      AN #s_Receive_Data_Outf.Itm_Data.Process_1.Screening_Not_Required;
      A #s_Receive_Data_Outf.Itm_Data.HBS_Record.PEN_Process_1.Result_Pending;
      A(;
      L "DB_HBS_List".HBS[#s_Receive_Data_Outf.Itm_Data.LNK_Record.HBS].LNK;// nlpcanh //#s_Receive_Data_Outf.Itm_Data.HBS_Record.PEN_General.HBA_LNK
      L #s_Receive_Data_Outf.Itm_Data.LNK;
      ==I;
      );
      A(;
      L #s_Receive_Data_Outf.Itm_Data.HBS_Record.PEN_Process_1.Screen_Result.Pseudo_ID;
      L #s_ISD_ID_Tracking.Data_10.BHS_Pseudo_Bag_ID;
      ==D;
      );
      S #s_Receive_Data_Outf.Itm_Data.Process_1.Screening_Pending;
      S #s_Receive_Data_Outf.Screening_Pending;// If a certain process contains the pseudo which is sent by the EDS, while "result expected": item is pending

IB01:      A #s_Receive_Data_Outf.EDS_Tracking.Trk_Lost_Result_Pending;
      JCN IB99;
//// [CPH] If lost in tracking inside the machine, do not expect/accept any further decisions
////      SET
////      S     #s_Receive_Data_Outf.Itm_Data.Process_1.Screening_Pending
////      S     #s_Receive_Data_Outf.Screening_Pending

IB99:      NOP 0;
NETWORK
TITLE = JA: Update GENERAL local records (HBS/LIC) at outfeed
//Local records will be updated to reflect the current bag status.
      A #s_OS_Receive_Bag_Data;// Bag tracking was restored (outfeed)
      A #s_Receive_Data_Outf.Tracking_Restored;// Check HBS record
      JCN JA99;

      L #i_HBS_ID;
      T #t_Last_Location;

      CALL "FC_Write_Dint_Record"
      (  i_Record_Number             := #s_Receive_Data_Outf.Itm_Data.LNK_Record.ECS ,
         i_P_DINT_Record             := "DB_UDT_ECS_Record".CIR.Last_Location ,
         i_DB                        := "DB_ECS_List" ,
         i_DINT                      := #t_Last_Location ,
         i_DB_Event_Num              := #t_DB_Event_Num_Object
      );

      A #s_Receive_Data_Outf.Screening_Pending;
      JCN JA99;

      A #s_Receive_Data_Outf.HBS_Record_Present;
      JCN JA01;

      CALL "FC_Read_ANY_Record"
      (  i_Record_Number             := #s_Receive_Data_Outf.Itm_Data.LNK_Record.HBS ,
         i_ANY_Data_Record           := "DB_UDT_HBS_Record".PEN_General ,
         i_ANY_Data                  := #s_Receive_Data_Outf.Itm_Data.HBS_Record.PEN_General ,
         i_DB                        := "DB_HBS_List" ,
         i_DB_Event_Num              := #t_DB_Event_Num_Object
      );

      JU JA99;

JA01:      CALL "FC_Generator_LNK"
      (  i_LNK                       := #s_Receive_Data_Outf.Itm_Data.LNK ,
         i_DB_List                   := #t_DB_HBS_List_Num ,
         i_Default_Record            := #i_Default_Record_Outf ,
         i_DB_Event_Num              := #t_DB_Event_Num_Object ,
         o_LNK                       := #t_INT_not_used
      );

      CALL "FC_Read_Int_Record"
      (  i_Record_Number             := #s_Receive_Data_Outf.Itm_Data.LNK ,
         i_P_INT_Record              := "DB_UDT_LNK_Record".HBS ,
         i_DB                        := "DB_LNK_List" ,
         i_DB_Event_Num              := #t_DB_Event_Num_Object ,
         o_INT                       := #s_Receive_Data_Outf.Itm_Data.LNK_Record.HBS
      );

      CALL "FC_Read_ANY_Record"
      (  i_Record_Number             := #s_Receive_Data_Outf.Itm_Data.LNK_Record.HBS ,
         i_ANY_Data_Record           := "DB_UDT_HBS_Record" ,
         i_ANY_Data                  := #s_Receive_Data_Outf.Itm_Data.HBS_Record ,
         i_DB                        := "DB_HBS_List" ,
         i_DB_Event_Num              := #t_DB_Event_Num_Object
      );

      L #s_Receive_Data_Outf.Itm_Data.LNK_Record.HBS;
      L 0;
      >I;
      S #s_Receive_Data_Outf.HBS_Record_Present;
      JCN JA99;// Creation succeeded

      SET;
      R #s_Receive_Data_Outf.Itm_Data.HBS_Record.PEN_General.Item_Lost;
      S #s_Receive_Data_Outf.Init_HBS_Record;

      L 0;
      T #s_Receive_Data_Outf.Itm_Data.HBS_Record.PEN_General.AreaID_Receive;

      CALL "FC_Write_ANY_Record"// Attach to bag
      (  i_Record_Number             := #s_Receive_Data_Outf.Itm_Data.LNK_Record.HBS ,
         i_ANY_Data_Record           := "DB_UDT_HBS_Record".PEN_General ,
         i_ANY_Data                  := #s_Receive_Data_Outf.Itm_Data.HBS_Record.PEN_General ,
         i_DB                        := "DB_HBS_List" ,
         i_DB_Event_Num              := #t_DB_Event_Num_Object
      );

      A #s_Receive_Data_Outf.New_LNK_Created;
      JCN JA99;// If new LNK with HBS was created: store HBS number in lookup table

      L #s_EDS_Pseudo_Lookup.Write_Position_Lookup_T;
      JL JA10;
      JU JA11;
      JU JA12;
      JU JA13;
      JU JA14;
      JU JA15;
JA10:      JU JA99;
JA11:      L #s_Receive_Data_Outf.Itm_Data.LNK_Record.HBS;
      T #s_EDS_Pseudo_Lookup.HBS_Lookup_Table[0];
      JU JA20;
JA12:      L #s_Receive_Data_Outf.Itm_Data.LNK_Record.HBS;
      T #s_EDS_Pseudo_Lookup.HBS_Lookup_Table[1];
      JU JA20;
JA13:      L #s_Receive_Data_Outf.Itm_Data.LNK_Record.HBS;
      T #s_EDS_Pseudo_Lookup.HBS_Lookup_Table[2];
      JU JA20;
JA14:      L #s_Receive_Data_Outf.Itm_Data.LNK_Record.HBS;
      T #s_EDS_Pseudo_Lookup.HBS_Lookup_Table[3];
      JU JA20;
JA15:      L #s_Receive_Data_Outf.Itm_Data.LNK_Record.HBS;
      T #s_EDS_Pseudo_Lookup.HBS_Lookup_Table[4];

JA20:      L #s_EDS_Pseudo_Lookup.Write_Position_Lookup_T;
      L 1;
      +I;
      T #s_EDS_Pseudo_Lookup.Write_Position_Lookup_T;

      L #s_EDS_Pseudo_Lookup.Write_Position_Lookup_T;
      L 4;
      >I;
      JCN JA99;

      L 0;
      T #s_EDS_Pseudo_Lookup.Write_Position_Lookup_T;
JA99:      NOP 0;
NETWORK
TITLE = JB: Update PROCESS_1 local records (HBS/LIC) at outfeed
      A #s_OS_Receive_Bag_Data;
      JCN JB99;

      A #s_Receive_Data_Outf.New_LNK_Created;
      AN #s_Receive_Data_Outf.LIC_Missing;
      JCN JB01;// If LIC is available and a new records was generated: attach pseudo, else: continue HBS record update

      CALL "FC_Write_Dint_Record"// Write pseudo to LIC
      (  i_Record_Number             := #s_Receive_Data_Outf.Itm_Data.LNK_Record.LIC ,
         i_P_DINT_Record             := "DB_UDT_LIC_Record".BIR.Process_1.Pseudo_ID ,
         i_DB                        := "DB_LIC_List" ,
         i_DINT                      := #s_PseudoId_To_Use_At_Exit , //#s_ISD_ID_Tracking.Data_10.BHS_Pseudo_Bag_ID
         i_DB_Event_Num              := #t_DB_Event_Num_Object
      );

JB01:      A #s_Receive_Data_Outf.Screening_Pending;
      A #s_Receive_Data_Outf.HBS_Record_Present;
      JCN JB99;// If new data prepared: create records and check if HBS record update is required

      A #s_Receive_Data_Outf.Init_HBS_Record;
      JCN JB02;

      SET;
      R #s_Receive_Data_Outf.Itm_Data.HBS_Record.PEN_Process_1.Machine_Result_Rcvd;
      R #s_Receive_Data_Outf.Itm_Data.HBS_Record.PEN_Process_1.Operator_Result_Rcvd;
      R #s_Receive_Data_Outf.Itm_Data.HBS_Record.PEN_Process_1.Result_Pending;
      R #s_Receive_Data_Outf.Itm_Data.HBS_Record.PEN_Process_1.Update_Send;
      R #s_Receive_Data_Outf.Itm_Data.HBS_Record.PEN_Process_1.Resend_Required;
      R #s_Receive_Data_Outf.Itm_Data.HBS_Record.PEN_Process_1.Force_Rejected;

      L 0;
      T #s_Receive_Data_Outf.Itm_Data.HBS_Record.PEN_General.TRA_LNK;
      T #s_Receive_Data_Outf.Itm_Data.HBS_Record.PEN_General.HBA_LNK;

      CALL "FC_Any_To_Adress"
      (  i_ANY_Data                  := #s_Receive_Data_Outf.Itm_Data.HBS_Record.PEN_General.Bag_Status ,
         o_Adress                    := #t_adress   //Determine the adress to Bag_Status
      );

      L #t_adress;
      SLD 3;// Shift bytes to make pointer to last entry
      LAR2;// Pointer to Bag_Status

      L 0;
      T DIW[ AR2, P#0.0];// Clear Bag_Status

      L DINT#0;
      T #s_Receive_Data_Outf.Itm_Data.HBS_Record.PEN_Process_1.Screen_Result.Pseudo_ID;
      T #s_Receive_Data_Outf.Itm_Data.HBS_Record.PEN_Process_1.ID_Screening;

JB02:      A #s_Receive_Data_Outf.Itm_Data.Process_1.Screening_Pending;
      JCN JB90;// If bag is about te be screened: fill in HBS record

      SET;
      S #s_Receive_Data_Outf.Itm_Data.HBS_Record.PEN_Process_1.Result_Pending;

      CALL RD_SYS_T// Write timestamp
      {date_type := 'Date_And_Time'}
      (  RET_VAL                     := #t_INT_not_used ,
         OUT                         := #s_Receive_Data_Outf.Itm_Data.HBS_Record.PEN_Process_1.Timestamp_screening
      );

      L #s_Receive_Data_Outf.Itm_Data.LNK;// Write LNK
      T #s_Receive_Data_Outf.Itm_Data.HBS_Record.PEN_General.HBA_LNK;

      L #i_HBO_ID;// Write screening machine ID
      T #s_Receive_Data_Outf.Itm_Data.HBS_Record.PEN_Process_1.ID_Screening;

      L #i_Local_Destination;
      T #s_Receive_Data_Outf.Itm_Data.HBS_Record.PEN_Process_1.EDS_Destination;

      CALL "FC_Read_ANY_Record"// Sync already present process data
      (  i_Record_Number             := #s_Receive_Data_Outf.Itm_Data.LNK_Record.LIC ,
         i_ANY_Data_Record           := "DB_UDT_LIC_Record".BIR.Process_1 ,
         i_ANY_Data                  := #s_Receive_Data_Outf.Itm_Data.HBS_Record.PEN_Process_1.Screen_Result ,
         i_DB                        := "DB_LIC_List" ,
         i_DB_Event_Num              := #t_DB_Event_Num_Object
      );

      L #s_PseudoId_To_Use_At_Exit;//#s_ISD_ID_Tracking.Data_10.BHS_Pseudo_Bag_ID// Write pseudo
      T #s_Receive_Data_Outf.Itm_Data.HBS_Record.PEN_Process_1.Screen_Result.Pseudo_ID;

      CALL "FC_Write_ANY_Record"// Attach to bag
      (  i_Record_Number             := #s_Receive_Data_Outf.Itm_Data.LNK_Record.HBS ,
         i_ANY_Data_Record           := "DB_UDT_HBS_Record".PEN_Process_1 ,
         i_ANY_Data                  := #s_Receive_Data_Outf.Itm_Data.HBS_Record.PEN_Process_1 ,
         i_DB                        := "DB_HBS_List" ,
         i_DB_Event_Num              := #t_DB_Event_Num_Object
      );

      L "DB_LNK_List".LNK[#s_Receive_Data_Outf.Itm_Data.LNK].HBS;
      T #t_LIC;

      L "DB_HBS_List".HBS[#s_Receive_Data_Outf.Itm_Data.LNK_Record.HBS].PEN_General.PEN_ID;
      T #t_PEN_ID;

      CALL MOVE
      {value_type := 'Variant'}
      (  IN                          := "DB_HBS_List".HBS[#t_LIC].PEN_Process_1 ,
         OUT                         := "DB_Pending_Record".THIS[#t_PEN_ID].PEN.PEN_Process_1
      );
      JU JB99;

JB90:      AN #s_Receive_Data_Outf.Itm_Data.HBS_Record.PEN_Process_1.Result_Pending;
      AN #s_Receive_Data_Outf.Itm_Data.HBS_Record.PEN_Process_2.Result_Pending;
      AN #s_Receive_Data_Outf.Itm_Data.HBS_Record.PEN_Process_3.Result_Pending;
      AN #s_Receive_Data_Outf.Itm_Data.HBS_Record.PEN_Process_4.Result_Pending;
      AN #s_Receive_Data_Outf.Itm_Data.HBS_Record.PEN_Process_5.Result_Pending;
      JCN JB99;
//If item is not screen pending, deassign the HBS and pending record
      CALL "FC_PEN_Deassign"
      (  i_PEN_ID                    := #t_PEN_ID
      );

      L 0;
      T "DB_LNK_List".LNK[#s_Receive_Data_Outf.Itm_Data.LNK].HBS;
      T "DB_HBS_List".HBS[#s_Receive_Data_Outf.Itm_Data.LNK_Record.HBS].LNK;
JB99:      NOP 0;

NETWORK
TITLE = KA: Handle data receiving errors and statisticals at outfeed
//Check incoming data to detect errors
      AN #s_Receive_Data_Outf.Tracking_Restored;// Error occured while trying to restore tracking
      O #s_Receive_Data_Outf.Lost_In_Tracking;
      A #s_OS_Receive_Bag_Data;
      AN #i_Allow_Unexpected_Data;
      JCN KA01;// Tracking NOK. Increment lost count

      L #s_Receive_Data_Outf.Succ_Tracking_Lst_Cnt;
      L 1;
      +I;
      T #s_Receive_Data_Outf.Succ_Tracking_Lst_Cnt;

      AN #s_Receive_Data_Outf.Tracking_Restored;
      JCN KA01;// Data matching failed: log event

      CALL "FC_Write_Event"// 3201 Log_Text := 'Screening: Received unknown BagID from HBS'
      (  i_Message_ID                := 3201 ,
         i_Event_value               := #s_Receive_Data_Outf.Itm_Data.LNK ,
         i_DB_Event_Num              := #t_DB_Event_Num_Object ,
         o_Return_Value              := #t_INT_not_used
      );

KA01:      A #s_Receive_Data_Outf.Tracking_Restored;
      AN #s_Receive_Data_Outf.New_LNK_Created;
      A #s_OS_Receive_Bag_Data;
      O(;
      A #i_CMD_Reset;
      A #o_ST_Succ_Unexp_Data;
      );
      JCN KA02;// Tracking OK. Reset lost count

      L 0;
      T #s_Receive_Data_Outf.Succ_Tracking_Lst_Cnt;

KA02:      L #i_HBO_Settings.Code_Req_Position_Outf;
      L #i_HBO_Settings.Srch_Dwn_Window;
      -I;
      JPZ KA03;
      L 0;
KA03:      T #t_Position;

      L #i_HBO_Settings.Srch_Up_Window;
      L #i_HBO_Settings.Srch_Dwn_Window;
      +I;
      T #t_Window;

      CALL "FC_PLT_Srch_Inf_Up"// Search for LNK number in PLT DB
      (  i_DB_PLT_Num                := #s_DB_PLT_Num_Outfeed ,
         i_Position                  := #t_Position ,
         i_Window                    := #t_Window ,
         i_Info                      := 1 ,
         o_Position                  := #t_INT_not_used ,
         o_Info                      := #t_INT_not_used ,
         o_LNK                       := #t_INT_not_used ,
         o_DB_PLT_Num                := #t_INT_not_used ,
         o_Number_Items_Found        := #s_Number_Of_Items_Found
      );

      L #s_Number_Of_Items_Found;
      L 0;
      >I;
      = #t_Bag_In_Upd_Window_Outf;

      A #s_OS_Receive_Bag_Data;
      A #t_Bag_In_Upd_Window_Outf;
      S #s_EDS_Data_Received;

      A #t_Bag_In_Upd_Window_Outf;
      FN #s_FN_Bag_In_Upd_Win_Outf;
      AN #s_EDS_Data_Received;
      AN #i_IO_Transport_Mode;
      JCN KA04;// If a bag left the update window while no data was received: Log

      CALL "FC_Write_Event"
      (  i_Message_ID                := 3214 , // Screening: No EDS data received for item in upd window at outfeed
         i_Event_value               := 0 , // LNK still unknown due to black box
         i_DB_Event_Num              := #t_DB_Event_Num_Object ,
         o_Return_Value              := #t_INT_not_used
      );

      L #s_Receive_Data_Outf.Succ_No_Data;
      L 1;
      +I;
      T #s_Receive_Data_Outf.Succ_No_Data;

KA04:      AN #t_Bag_In_Upd_Window_Outf;
      R #s_EDS_Data_Received;

      A #i_CMD_Reset;
      A #o_ST_Succ_No_Data;
      O #s_OS_Receive_Bag_Data;
      JCN KA05;// Reset successive no data when new data is received

      L 0;
      T #s_Receive_Data_Outf.Succ_No_Data;

KA05:      AN #i_Test_Mode_Active;
      JCN KA90;// Don't count statisticals in test mode

      A #s_OS_Receive_Bag_Data;
      A #s_Receive_Data_Outf.EDS_Tracking.Positively_Tracked;
      JCN KA07;

      L #s_Statisticals.Tracking.Positively_Tracked;
      L 1;
      +I;
      JP KA06;
      L 1;
KA06:      T #s_Statisticals.Tracking.Positively_Tracked;

KA07:      A #s_OS_Receive_Bag_Data;
      A #s_Receive_Data_Outf.EDS_Tracking.Trk_Lost_Result_Pending;
      JCN KA09;

      L #s_Statisticals.Tracking.Trk_Lost_Result_Pending;
      L 1;
      +I;
      JP KA08;
      L 1;
KA08:      T #s_Statisticals.Tracking.Trk_Lost_Result_Pending;

KA09:      A #s_OS_Receive_Bag_Data;
      A #s_Receive_Data_Outf.EDS_Tracking.Trk_Lost_No_Result;
      JCN KA90;

      L #s_Statisticals.Tracking.Trk_Lost_No_Result;
      L 1;
      +I;
      JP KA10;
      L 1;
KA10:      T #s_Statisticals.Tracking.Trk_Lost_No_Result;

KA90:      A #i_CMD_Reset;
      R #o_ST_Succ_Unexp_Data;
      R #o_ST_Succ_No_Data;

      A(;
      L #i_CFG_Num_Unex_Data_Er;
      L #s_Receive_Data_Outf.Succ_Tracking_Lst_Cnt;
      <=I;
      );
      A(;
      L #i_CFG_Num_Unex_Data_Er;
      L 0;
      <>I;
      );
      S #o_ST_Succ_Unexp_Data;

      A(;
      L #i_CFG_Num_No_Data_Er;
      L #s_Receive_Data_Outf.Succ_No_Data;
      <=I;
      );
      A(;
      L #i_CFG_Num_No_Data_Er;
      L 0;
      <>I;
      );
      S #o_ST_Succ_No_Data;
NETWORK
TITLE = LA: Clean up non tracking DB at outfeed
//Non tracking PLT DB clean up
//- Upon receival of new data: remove received item if tracking is restored and
//remove data which got lost according to the FIFO principle
//- When the EDS reports to be empty: clean up entire PLT DB
      A #i_IO_EDS_Bag_In_Process;
      O;
      A #s_Bag_In_Process_Delayed;
      A(;
      A #t_OS_Physical_Handover;
      ON #i_IO_HBS_Conv_Run_Feedback;// nlpcanh - 16-02-2026 - keep data while HBS stopped
      );
      = #t_IO_Bag_In_Process;// Prevent clear PLT due to signal delays (prevent race condition)

      CALL "FC_Off_Dly_T_0.1s"
      (  i_Start                     := #t_IO_Bag_In_Process ,
         i_Enable_Dly                := TRUE ,
         i_Time_Value                := 70 , //nlpcanh - 16-02-2026 - #i_IO_EDS_Bag_In_Process is dropped after bag out of x-ray beam // 15
         i_Current_Value             := #s_IO_Bag_In_Process_Cnt ,
         o_Status                    := #s_Bag_In_Process_Delayed ,
         o_Current_Value             := #s_IO_Bag_In_Process_Cnt
      );

      AN #s_Bag_In_Process_Delayed;
      FP #s_FP_EDS_Empty;
      = #s_OS_EDS_Empty;

      AN #i_Available_IO;// Clear on comms loss
      AN #i_IO_EDS_Bag_In_Process;
      O #i_Comm_Error;
      A(;
      L #o_Nr_Items;
      L 0;
      >I;
      );
      O #s_OS_EDS_Empty;// Clear when EDS reports "empty"
      O "M_First_Scan";// Clear on first scan
      = #s_Clear_Non_Trk_PLT_DB;

//in NW IA: Receive data from EDS (restore tracking) at outfeed --> how it works:
//--> LNK of the bag is found in shadow PLT, PLT DB nr value (inside of LNK record) is overwritten with TRS05 value.
//--> This is how LNK is moved from TRS03 (shadow PLT) to TRS05 PLT.

//since LNK is moved from shadow PLT to TRS05 in the network IA, below 4 variables are commented.
//there is no need to clear the item at the end of the TRS03 PLT DB, because that item is transferred already at this point of time.
//Executing network below based on #s_OS_Receive_Bag_Data or #s_Receive_Data_Outf.Tracking_Restored will clear 2nd item, which is still inside of the HBZ.
//A     #s_OS_Receive_Bag_Data
//A     #s_Receive_Data_Outf.Tracking_Restored
//AN    #s_Receive_Data_Outf.New_LNK_Created
//O     #t_Clear_Non_Trk_PLT_DB

      A #s_Clear_Non_Trk_PLT_DB;
      JCN LA02;// If tracking data is restored using shadow PLT data: clean-up shadow PLT

LA01:      CALL "FC_PLT_Srch_Inf_Up"
      (  i_DB_PLT_Num                := #t_DB_PLT_Num_Non_Trk ,
         i_Position                  := 0 ,
         i_Window                    := #t_PLT_Non_Trk_Length ,
         i_Info                      := 1 ,
         o_Position                  := #t_Position ,
         o_Info                      := #t_INT_not_used ,
         o_LNK                       := #t_LNK_Found ,
         o_DB_PLT_Num                := #t_INT_not_used ,
         o_Number_Items_Found        := #t_Num_Items_Found
      );

      L #t_Num_Items_Found;
      L 0;
      <>I;
      JCN LA02;

      CALL "FC_PLT_Clr_Position"
      (  i_DB_PLT_Num                := #t_DB_PLT_Num_Non_Trk ,
         i_Position                  := #t_Position ,
         i_Info_Physical             := 1 ,
         i_DB_Event_Num              := -1   //Events not reported
      );

      A(;
      L #t_LNK_Found;
      L #s_Receive_Data_Outf.Itm_Data.LNK;
      ==I;// IF LNK found was not the one which was received from the EDS OR EDS indicates it has no items in tracking
      );// Current (found) item is consider lost according to the FIFO principle -> deregister
      A #s_OS_Receive_Bag_Data;
      = #t_LNK_Clrd_Non_Trk_DB;


      AN #s_Clear_Non_Trk_PLT_DB;
      A #t_LNK_Clrd_Non_Trk_DB;// If received LNK is found in non tracking PLT DB while EDS not reporting empty: End cleanup,
      JC LA02;// else: Continue

      A #s_Clear_Non_Trk_PLT_DB;
      A #t_LNK_Clrd_Non_Trk_DB;// If received LNK is found in non tracking PLT DB while EDS reporting empty: Also remove other records,
      JC LA01;// else: Deregister current item since it is considered lost

      CALL "FC_Read_Int_Record"
      (  i_Record_Number             := #t_LNK_Found ,
         i_P_INT_Record              := "DB_UDT_LNK_Record".ECS ,
         i_DB                        := "DB_LNK_List" ,
         i_DB_Event_Num              := #t_DB_Event_Num_Object ,
         o_INT                       := #t_ECS
      );

      CALL "FC_Write_BOOL_Record"
      (  i_Record_Number             := #t_ECS ,
         i_P_BOOL_Record             := "DB_UDT_ECS_Record".CIR.Expected_Item ,
         i_DB                        := "DB_ECS_List" ,
         i_BOOL                      := FALSE ,
         i_DB_Event_Num              := #t_DB_Event_Num_Object
      );

      CALL "FC_Write_BOOL_Record"
      (  i_Record_Number             := #t_ECS ,
         i_P_BOOL_Record             := "DB_UDT_ECS_Record".CIR.Unexpected_Item ,
         i_DB                        := "DB_ECS_List" ,
         i_BOOL                      := TRUE ,
         i_DB_Event_Num              := #t_DB_Event_Num_Object
      );

      CALL "FC_Write_BOOL_Record"
      (  i_Record_Number             := #t_ECS ,
         i_P_BOOL_Record             := "DB_UDT_ECS_Record".CIR.Hand_Over ,
         i_DB                        := "DB_ECS_List" ,
         i_BOOL                      := FALSE ,
         i_DB_Event_Num              := #t_DB_Event_Num_Object
      );

      CALL "FC_Write_Event"// Send DeregisterPackage (1206)
      (  i_Message_ID                := 1206 ,
         i_Event_value               := #t_LNK_Found ,
         i_DB_Event_Num              := #t_DB_Event_Num_Section ,
         o_Return_Value              := #t_INT_not_used
      );

      JU LA01;// LOOP: Check if next record contains the correct LNK number OR loop till empty
LA02:      NOP 0;
///   A     #i_IO_EDS_Bag_In_Process
/// nlpcanh - 18-02-2026 - Bag_In_Process signal is too short, only active when bag under the x-ray beam.
      O #s_Bag_In_Process_Delayed;
      O(;
      L #o_Nr_Items;
      L 0;
      >I;
      );
///
      = #o_ST_Items;

NETWORK
TITLE = MA: Detect the receival of new decision data
      AN #i_IO_Decision_Available;
      R #s_Decision_Data.Sec_Bag_Dec_Processed;

      CALL "FC_On_Dly_T_0.1s"
      (  i_Start                     := #i_IO_Decision_Available ,
         i_Enable_Dly                := TRUE ,
         i_Time_Value                := 2 ,
         i_Current_Value             := #s_IO_Rcve_Dec_Dly_Cnt ,
         o_Status                    := #t_IO_Receive_Dec_Dly ,
         o_Current_Value             := #s_IO_Rcve_Dec_Dly_Cnt
      );

      A #t_IO_Receive_Dec_Dly;
      AN #s_OS_Receive_Bag_Data;// If decision available in exit bag data, process first
      AN #s_Decision_Data.Sec_Bag_Dec_Processed;// Process every security bag decision only once
      FP #s_FP_New_Decision_Avail;
      S #s_Decision_Data.Sec_Bag_Dec_Processed;
      = #s_OS_New_Decision_Avail;

      A #s_Decision_Data.Sec_Bag_Dec_Processed;
      = #o_IO_Ack_Sec_Bag_Data;// Acknowledge

      A #s_OS_New_Decision_Avail;
      O #s_OS_Receive_Bag_Data;
      JCN MA99;// If new decision data available (exit bag decision OR security bag decision): process it

      CALL "FC_Read_ANY_Record"
      (  i_Record_Number             := 0 ,
         i_ANY_Data_Record           := "DB_UDT_LNK_Record" ,
         i_ANY_Data                  := #s_Decision_Data.Itm_Data.LNK_Record ,
         i_DB                        := "DB_LNK_List" ,
         i_DB_Event_Num              := #t_DB_Event_Num_Object
      );

      CALL "FC_Read_ANY_Record"
      (  i_Record_Number             := 0 ,
         i_ANY_Data_Record           := "DB_UDT_HBS_Record" ,
         i_ANY_Data                  := #s_Decision_Data.Itm_Data.HBS_Record ,
         i_DB                        := "DB_HBS_List" ,
         i_DB_Event_Num              := #t_DB_Event_Num_Object
      );

      SET;
      R #s_Decision_Data.Valid_LNK_Available;
      R #s_Decision_Data.Inval_LNK_Pseudo_Lookup;
      R #s_Decision_Data.LIC_Missing;
      R #s_Decision_Data.Send_Package_Report;
      R #s_Decision_Data.Package_Report_Sent;
      R #s_Decision_Data.No_Decision_Expected;

      L DINT#0;
      T #s_Decision_Data.Itm_Data.Pseudo;

      L 0;
      T #s_Decision_Data.Itm_Data.LNK;

      A #s_OS_Receive_Bag_Data;
      JCN MA01;// Load decision data from correct process (exit bag decision or security bag decision)

// Data from CH0 (at Exit of machine)
      L #s_ISD_ID_Tracking.Data_7.LNK;
      T #t_PEN_ID;
//Check PEN_ID is valid
      A(;
      L #t_PEN_ID;
      L 0;
      >I;
      );
      A(;
      L #t_PEN_ID;
      L "DB_PEN_List".Entries_Present;
      <=I;
      );
      JCN MA99;

      L #t_PEN_ID;
      T #s_Decision_Data.Itm_Data.PEN_ID;

      L "DB_Pending_Record".THIS[#t_PEN_ID].PEN_LNK;
      T #s_Decision_Data.Itm_Data.LNK;

      L #s_PseudoId_To_Use_At_Exit;//#s_ISD_ID_Tracking.Data_10.BHS_Pseudo_Bag_ID
      T #s_Decision_Data.Itm_Data.Pseudo;

      JU MA99;

// Data from CH1 (Decision)
MA01:      L #s_ISD_ID_Decision.Data_7.LNK;
      T #t_PEN_ID;
//Check PEN_ID is valid
      L #t_PEN_ID;
      L 0;
      <=I;
      O(;
      L #t_PEN_ID;
      L "DB_PEN_List".Entries_Present;
      >I;
      );
      R #s_OS_New_Decision_Avail;

      A #s_OS_New_Decision_Avail;
      JCN MA99;

      L #t_PEN_ID;
      T #s_Decision_Data.Itm_Data.PEN_ID;

      L "DB_Pending_Record".THIS[#t_PEN_ID].PEN_LNK;
      T #s_Decision_Data.Itm_Data.LNK;

      L #s_ISD_ID_Decision.Data_10.BHS_Pseudo_Bag_ID;
      T #s_Decision_Data.Itm_Data.Pseudo;

MA99:      NOP 0;
NETWORK
TITLE = MB: Receive PROCESS_1 EDS decision and find applicable item
//Map EDS decision to readable STATs and find the correct bagage item. Bagage
//item can be found using the LNK or by a pseudo lookup in the HBS records.
      NOP 0;
// Determine type of line
      L #i_CFG_Line_Type;
      L 1;
      ==I;
      = #t_LineType_L1_L2a_L2b;// Special OOG line - CPH T3A

      L #i_CFG_Line_Type;
      L 2;
      ==I;
      = #t_LineType_L1_L2;// L2 is last decision expected

      L #i_CFG_Line_Type;
      L 3;
      ==I;
      = #t_LineType_L1_L2_L3;// L3 is last decision expected

      SET;
      R #t_Decision_Is_L2a;
      R #t_Decision_Is_L2b;
      R #t_Decision_Is_L2;
      R #t_Decision_Is_L3;
      R #t_Disposition_range_L2;
      R #t_Disposition_range_L3;

// When decision received
      A #s_OS_New_Decision_Avail;
      O #s_OS_Receive_Bag_Data;
      JCN MB99;// If new decision data available (exit bag decision OR security bag decision): process it

      L 0;
      T #s_Decision_Data.Itm_Data.Process_1.EDS_Decision.Decision_Bag_Disposition;
      T #s_Decision_Data.Itm_Data.Process_1.Machine_Result_To_HL;
      T #s_Decision_Data.Itm_Data.Process_1.Operator_Result_To_HL;

      SET;
      R #s_Group0_Read;
      R #s_Group1_Read;

      SET;// Clear static data
      R #s_Decision_Data.Itm_Data.Process_1.EDS_Decision.No_Decision;//0 = No Decision (library)
      R #s_Decision_Data.Itm_Data.Process_1.EDS_Decision.Not_Analyzed;//RTT110: (Byte_1) 3 = Machine Analysis Error / Machine Mistrack
      R #s_Decision_Data.Itm_Data.Process_1.EDS_Decision.Decision_Pending;//RTT110: (Byte_1) 4 = Decision Pending
      R #s_Decision_Data.Itm_Data.Process_1.EDS_Decision.Cleared_Machine;//RTT110: (Byte_1) 1 = Machine Cleared
      R #s_Decision_Data.Itm_Data.Process_1.EDS_Decision.Rejected_Machine;//RTT110: (Byte_1) 2 = Machine Threat or Machine Shield Alarm
      R #s_Decision_Data.Itm_Data.Process_1.EDS_Decision.L2_L3_L4_Unknown;//RTT110: (Byte_2_3_4) = Unknown
      R #s_Decision_Data.Itm_Data.Process_1.EDS_Decision.L2_Operator_Cleared;
      R #s_Decision_Data.Itm_Data.Process_1.EDS_Decision.L2_Operator_Rejected;
      R #s_Decision_Data.Itm_Data.Process_1.EDS_Decision.L2_Operator_Timed_Out;
      R #s_Decision_Data.Itm_Data.Process_1.EDS_Decision.L2_Matrix_Timeout_Matrix_Error;
      R #s_Decision_Data.Itm_Data.Process_1.EDS_Decision.L3_Operator_Cleared;
      R #s_Decision_Data.Itm_Data.Process_1.EDS_Decision.L3_Operator_Rejected;
      R #s_Decision_Data.Itm_Data.Process_1.EDS_Decision.L3_Operator_Timed_Out;
      R #s_Decision_Data.Itm_Data.Process_1.EDS_Decision.L3_Matrix_Timeout_Matrix_Error;//RTT110: (Byte_1) 3 = Machine Analysis Error / Machine Mistrack
      R #s_Decision_Data.Itm_Data.Process_1.EDS_Decision.No_Scan_Bag_RTT;//RTT110: (Byte_1) 9 = No Scan Bag
      R #s_Decision_Data.Itm_Data.Process_1.EDS_Decision.EDS_Error;
      R #s_Decision_Data.Itm_Data.Process_1.EDS_Decision.Forced_Reject;//NA for RTT110. ONLY in FB_HBO_XCT it is set. Disposition = 7.
      R #s_Decision_Data.Itm_Data.Process_1.EDS_Decision.Obvious_Threat;//NA for RTT110. It is purely Smiths status.
      S #s_Decision_Data.Itm_Data.Process_1.No_Decision_Expected;

      A #s_Receive_Data_Outf.New_LNK_Created;//changed, does not exist in 2024 library
      R #s_Decision_Data.Itm_Data.Process_1.No_Decision_Expected;//changed, does not exist in 2024 library

      A #s_OS_Receive_Bag_Data;
      JCN MB05;// Load decision data from correct process (exit bag decision or security bag decision)

// Read disposition

//   In a rare case scenario CH0 and CH1 can be activated at the same time for the same bag.
//     CH0 contains old info, known when Handover started.
//     CH1 contains new decision, made availabe during handover.
//   For this case we are comparing the LNK from both channels to understand if it is the same bag.
      L #s_ISD_ID_Tracking.Data_7.LNK;// CH0 (disposition at exit)
      L #s_ISD_ID_Decision.Data_7.LNK;// CH1 (disposition after exit)
      ==I;
      A #i_IO_Receive_Data_Outf;
      A #i_IO_Decision_Available;
      = #s_Simultaneous_Decisions_CH0_CH1;

      AN #s_Simultaneous_Decisions_CH0_CH1;
      JCN MB05;// If decision at EDS exit is present in both channels for same bag, then use CH1

// Get disposition and security routing from --CH0--
      L 0;
      L #s_ISD_ID_Tracking.Data_9.Group1_Disp_Operator_P1;
      <>I;
      S #s_Group1_Read;
      JC MB02;
      L #s_ISD_ID_Tracking.Data_9.Group0_Disp_Machine_P1;
MB02:      T #s_Decision_Data.Itm_Data.Process_1.EDS_Decision.Decision_Bag_Disposition;

      AN #s_Group1_Read;
      S #s_Group0_Read;

      L #s_ISD_ID_Tracking.Data_3.Security_Routing_Req;// Read used security routing from CH0
      T #s_Decision_Data.Itm_Data.Process_1.Security_Routing;
      JU MB11;

// Get disposition and security routing from --CH1--
MB05:      L 0;
      L #s_ISD_ID_Decision.Data_9.Group1_Disp_Operator_P1;
      <>I;
      S #s_Group1_Read;
      JC MB08;
      L #s_ISD_ID_Decision.Data_9.Group0_Disp_Machine_P1;
MB08:      T #s_Decision_Data.Itm_Data.Process_1.EDS_Decision.Decision_Bag_Disposition;

      AN #s_Group1_Read;
      S #s_Group0_Read;

      L #s_ISD_ID_Decision.Data_3.Security_Routing_Req;// Read used security routing from CH1
      T #s_Decision_Data.Itm_Data.Process_1.Security_Routing;

// CPH: Determine decision Level (when in OOG line, then L1+L2a+L2b, so further down L3 needs to be translated to L2b)
MB11:      A(;
      L #s_Decision_Data.Itm_Data.Process_1.EDS_Decision.Decision_Bag_Disposition;
      L 10;
      >I;
      );
      A(;
      L #s_Decision_Data.Itm_Data.Process_1.EDS_Decision.Decision_Bag_Disposition;
      L 20;
      <I;
      );
      = #t_Disposition_range_L2;

      A(;
      L #s_Decision_Data.Itm_Data.Process_1.EDS_Decision.Decision_Bag_Disposition;
      L 20;
      >I;
      );
      A(;
      L #s_Decision_Data.Itm_Data.Process_1.EDS_Decision.Decision_Bag_Disposition;
      L 30;
      <I;
      );
      = #t_Disposition_range_L3;

      A #t_LineType_L1_L2a_L2b;
      A #s_Group1_Read;
      A #t_Disposition_range_L2;
      S #t_Decision_Is_L2a;// L2a

      A #t_LineType_L1_L2a_L2b;
      A #s_Group1_Read;
      A #t_Disposition_range_L3;
      S #t_Decision_Is_L2b;// L2b

      A #t_LineType_L1_L2;
      O #t_LineType_L1_L2_L3;
      A #s_Group1_Read;
      A #t_Disposition_range_L2;
      S #t_Decision_Is_L2;// L2

      A #t_LineType_L1_L2_L3;
      A #s_Group1_Read;
      A #t_Disposition_range_L3;
      S #t_Decision_Is_L3;// L3

// Evaluate disposition

MB15:      L 0;// 0=No decision on current process
      L #s_Decision_Data.Itm_Data.Process_1.EDS_Decision.Decision_Bag_Disposition;
      ==I;
      S #s_Decision_Data.Itm_Data.Process_1.EDS_Decision.No_Decision;
      JC MB20;

//EDS results called L2_Unknown, L3_Unknown, L4_Unknown will have Disposition=3, but on different bytes.
//Byte_1 = 3 (Machine Analysis Error / Machine Mistrack)
//Byte_2/3/4 = 3 (L2, L3, L4 Unknown)
      L 3;// 3=(Machine Analysis Error / Machine Mistrack)
      L #s_Decision_Data.Itm_Data.Process_1.EDS_Decision.Decision_Bag_Disposition;
      ==I;
      A #s_Group0_Read;
      S #s_Decision_Data.Itm_Data.Process_1.EDS_Decision.EDS_Error;
      JC MB20;

      L 3;// 3=(L2, L3, L4 Operator Unknown)
      L #s_Decision_Data.Itm_Data.Process_1.EDS_Decision.Decision_Bag_Disposition;
      ==I;
      A #s_Group1_Read;
      S #s_Decision_Data.Itm_Data.Process_1.EDS_Decision.L2_L3_L4_Unknown;//= Bag_Status.Unknown (HL message = 5)
      JC MB20;

      L 4;// 4=Decision pending
      L #s_Decision_Data.Itm_Data.Process_1.EDS_Decision.Decision_Bag_Disposition;
      ==I;
      S #s_Decision_Data.Itm_Data.Process_1.EDS_Decision.Decision_Pending;
      JC MB20;

      L 9;// 9=No Scan bag
      L #s_Decision_Data.Itm_Data.Process_1.EDS_Decision.Decision_Bag_Disposition;
      ==I;
      S #s_Decision_Data.Itm_Data.Process_1.EDS_Decision.No_Scan_Bag_RTT;
      JC MB20;

      L 1                  ;//1=Machine Alarm -> No Decision
      L #s_Decision_Data.Itm_Data.Process_1.EDS_Decision.Decision_Bag_Disposition;
      ==I;
      A(;
      L #s_Decision_Data.Itm_Data.Process_1.Security_Routing;
      L 13;// "show all"
      ==I;// If special routing mode is to "show all" images to operators,
      )                        ;// and machine rejects the bag, then ignore machine decision.
      S #s_Decision_Data.Itm_Data.Process_1.EDS_Decision.Rejected_Machine;
      JC MB20;

      L 1;//1=Machine Alarm
      L #s_Decision_Data.Itm_Data.Process_1.EDS_Decision.Decision_Bag_Disposition;
      ==I;
      S #s_Decision_Data.Itm_Data.Process_1.EDS_Decision.Rejected_Machine;
      JC MB20;

      L 2                  ;//2=Machine Cleared -> No Decision
      L #s_Decision_Data.Itm_Data.Process_1.EDS_Decision.Decision_Bag_Disposition;
      ==I;
      A(;
      L #s_Decision_Data.Itm_Data.Process_1.Security_Routing;
      L 13;// "show all"
      ==I;// If special routing mode is to "show all" images to operators,
      );// and machine clears the bag, then ignore machine decision.
      S #s_Decision_Data.Itm_Data.Process_1.EDS_Decision.No_Decision;
      JC MB20;

      L 2;//2=Machine Cleared
      L #s_Decision_Data.Itm_Data.Process_1.EDS_Decision.Decision_Bag_Disposition;
      ==I;
      S #s_Decision_Data.Itm_Data.Process_1.EDS_Decision.Cleared_Machine;
      JC MB20;
// L2 Operator Dispositions
      L 11;//11=Operator Alarm
      L #s_Decision_Data.Itm_Data.Process_1.EDS_Decision.Decision_Bag_Disposition;
      ==I;
      S #s_Decision_Data.Itm_Data.Process_1.EDS_Decision.L2_Operator_Rejected;
      JC MB20;

      L 12;//12=Operator Cleared
      L #s_Decision_Data.Itm_Data.Process_1.EDS_Decision.Decision_Bag_Disposition;
      ==I;
      S #s_Decision_Data.Itm_Data.Process_1.EDS_Decision.L2_Operator_Cleared;
      JC MB20;

      L 15;//15=Operator Timeout
      L #s_Decision_Data.Itm_Data.Process_1.EDS_Decision.Decision_Bag_Disposition;
      ==I;
      S #s_Decision_Data.Itm_Data.Process_1.EDS_Decision.L2_Operator_Timed_Out;
      JC MB20;

      L 16;//16=L2 Matrix Timeout / Matrix Error
      L #s_Decision_Data.Itm_Data.Process_1.EDS_Decision.Decision_Bag_Disposition;
      ==I;
      S #s_Decision_Data.Itm_Data.Process_1.EDS_Decision.L2_Matrix_Timeout_Matrix_Error;
      JC MB20;

// L3 Operator Dispositions
      L 21;//21=Operator Alarm
      L #s_Decision_Data.Itm_Data.Process_1.EDS_Decision.Decision_Bag_Disposition;
      ==I;
      S #s_Decision_Data.Itm_Data.Process_1.EDS_Decision.L3_Operator_Rejected;
      JC MB20;

      L 22;//22=Operator Cleared
      L #s_Decision_Data.Itm_Data.Process_1.EDS_Decision.Decision_Bag_Disposition;
      ==I;
      S #s_Decision_Data.Itm_Data.Process_1.EDS_Decision.L3_Operator_Cleared;
      JC MB20;

      L 25;//25=Operator Timeout
      L #s_Decision_Data.Itm_Data.Process_1.EDS_Decision.Decision_Bag_Disposition;
      ==I;
      S #s_Decision_Data.Itm_Data.Process_1.EDS_Decision.L3_Operator_Timed_Out;
      JC MB20;

      L 26;//26=L3 Matrix Timeout / Matrix Error
      L #s_Decision_Data.Itm_Data.Process_1.EDS_Decision.Decision_Bag_Disposition;
      ==I;
      S #s_Decision_Data.Itm_Data.Process_1.EDS_Decision.L3_Matrix_Timeout_Matrix_Error;
      JC MB20;

      SET;// all other result are unknown
      S #s_Decision_Data.Itm_Data.Process_1.EDS_Decision.Not_Analyzed;
      R #s_Decision_Data.Itm_Data.Process_1.EDS_Decision.Cleared_Machine;
      R #s_Decision_Data.Itm_Data.Process_1.EDS_Decision.Rejected_Machine;

MB20:      AN #s_Decision_Data.No_Decision_Expected;
      JCN MB98;

      AN #s_Decision_Data.Valid_LNK_Available;
      JCN MB21;// Item already found, no data reload needed

      A(;
      L #s_Decision_Data.Itm_Data.LNK;
      L 0;
      >I;
      );
      JCN MB22;// If LNK is unknown by EDS, start lookup on pseudo ID

      L #s_Decision_Data.Itm_Data.PEN_ID;
      L "DB_PEN_List".Entries_Present;
      <=I;
      JCN MB98;// If LNK is not in expected range: Abort data attachment

      L "DB_Pending_Record".THIS[#s_Decision_Data.Itm_Data.PEN_ID].PEN_LNK;
      L 0;
      ==I;
      S #s_Decision_Data.No_Decision_Expected;

      AN #s_Decision_Data.No_Decision_Expected;
      JCN MB98;// No HBS record = no screening result expected

      L "DB_Pending_Record".THIS[#s_Decision_Data.Itm_Data.PEN_ID].PEN.LNK;
      L 0;
      >I;
      JCN MB21;

      CALL "FC_Read_ANY_Record"// Read entire LNK record
      (  i_Record_Number             := #s_Decision_Data.Itm_Data.LNK ,
         i_ANY_Data_Record           := "DB_UDT_LNK_Record" ,
         i_ANY_Data                  := #s_Decision_Data.Itm_Data.LNK_Record ,
         i_DB                        := "DB_LNK_List" ,
         i_DB_Event_Num              := #t_DB_Event_Num_Object
      );

MB21:      L #s_Decision_Data.Itm_Data.Pseudo;
      L "DB_Pending_Record".THIS[#s_Decision_Data.Itm_Data.PEN_ID].PEN.PEN_Process_1.Screen_Result.Pseudo_ID;
      ==D;
      JCN MB22;

      L #s_Decision_Data.Itm_Data.PEN_ID;
      L 0;
      >I;
      JCN MB22;

      L "DB_Pending_Record".THIS[#s_Decision_Data.Itm_Data.PEN_ID].PEN.PEN_Process_1.ID_Screening;
      L #i_HBO_ID;
      ==D;
      S #s_Decision_Data.Valid_LNK_Available;
      R #s_Decision_Data.Itm_Data.Process_1.No_Decision_Expected;
      JU MB98;

MB22:      AN #s_Decision_Data.Valid_LNK_Available;
      JCN MB98;

      AN #s_Decision_Data.Itm_Data.Process_1.No_Decision_Expected;//Security_Routing_Req = 12 from BHS to HBZ.
      JCN MB99;

      SET;
      S #s_Decision_Data.Inval_LNK_Pseudo_Lookup;

      L DINT#0;
      L #s_Decision_Data.Itm_Data.Pseudo;
      <>D;
      JCN MB98;// If no pseudo available: End bag lookup, else: lookup bag by pseudo

      CALL "FC_PEN_Srch_ID"
      (  i_Pseudo_ID                 := #s_Decision_Data.Itm_Data.Pseudo ,
         o_PEN_ID                    := #s_Decision_Data.Itm_Data.PEN_ID
      );

      L #s_Decision_Data.Itm_Data.PEN_ID;
      L 0;
      >I;
      JCN MB99;


MB50:      AN #s_Decision_Data.Valid_LNK_Available;
      JCN MB98;// If correct LNK not found yet, try next pseudo


MB98:      A #s_Decision_Data.Itm_Data.Process_1.No_Decision_Expected;
      O #s_Decision_Data.No_Decision_Expected;
      AN #s_Decision_Data.Itm_Data.Process_1.EDS_Decision.No_Decision;
//AN    #s_Decision_Data.Itm_Data.Process_1.EDS_Decision.Forced_Reject// NA for RTT110
      AN #s_Decision_Data.Itm_Data.Process_1.EDS_Decision.Not_Analyzed;//With LIC=0 EDS responds Not Analyzed
      JCN MB99;// Unable to find applicable item or item is not pending while decision is present: log event

      CALL "FC_Write_Event"// Screening: Unexpected decision from EDS
      (  i_Message_ID                := 3213 ,
         i_Event_value               := #s_ISD_ID_Decision.Data_7.LNK ,
         i_DB_Event_Num              := #t_DB_Event_Num_Object ,
         o_Return_Value              := #t_INT_not_used
      );

MB99:      NOP 0;

NETWORK
TITLE = NA: Upd. PROCESS_1 records (HBS/LIC) upon decision + PackageRep
//Update local bag records to match received decisions
      A #s_OS_New_Decision_Avail;
      O #s_OS_Receive_Bag_Data;
      A #s_Decision_Data.Valid_LNK_Available;
      JCN NA99;

      AN #s_Decision_Data.Itm_Data.Process_1.No_Decision_Expected;
      JCN NA99;// If no HBS record available: stop receival, else: process

      CALL MOVE
      {value_type := 'Variant'}
      (  IN                          := "DB_Pending_Record".THIS[#s_Decision_Data.Itm_Data.PEN_ID].PEN ,
         OUT                         := #s_Decision_Data.Itm_Data.HBS_Record
      );

      AN #s_Decision_Data.Itm_Data.HBS_Record.PEN_Process_1.Result_Pending;
      O #s_Decision_Data.Itm_Data.HBS_Record.PEN_General.Item_Lost;
      O(;
      L #s_Decision_Data.Itm_Data.HBS_Record.PEN_General.HBA_LNK;
      L #s_Decision_Data.Itm_Data.LNK;
      <>I;
      );
      S #s_Decision_Data.Itm_Data.Process_1.No_Decision_Expected;// No decision expected concluded by HBS record content

      L "DB_Pending_Record".THIS[#s_Decision_Data.Itm_Data.PEN_ID].PEN.LNK;
      L 0;
      ==I;
      S #s_Decision_Data.LIC_Missing;

      AN #s_Decision_Data.Itm_Data.Process_1.No_Decision_Expected;
      AN #s_Decision_Data.Itm_Data.Process_1.EDS_Decision.No_Decision;
      AN #s_Decision_Data.Itm_Data.Process_1.EDS_Decision.No_Scan_Bag_RTT;
      JCN NA20               ;// If process 1 decision expected and present: process, else: make sure PackageReport DB is empty

// Check if current bag has already been screened.
      A #s_Decision_Data.Itm_Data.HBS_Record.PEN_General.Bag_Status.NoDecision;
      O #s_Decision_Data.Itm_Data.HBS_Record.PEN_General.Bag_Status.Unknown;
      O #s_Decision_Data.Itm_Data.HBS_Record.PEN_General.Bag_Status.EDS_Error;
      = #t_Bag_ReScreening;

//This is Bag_Status clear routine after every new status received from the machine.
//Only 1 Bag_Status will be active at a time.
      SET;
      R #s_Decision_Data.Itm_Data.HBS_Record.PEN_General.Bag_Status.TimeOut;
      R #s_Decision_Data.Itm_Data.HBS_Record.PEN_General.Bag_Status.Unknown;
      R #s_Decision_Data.Itm_Data.HBS_Record.PEN_General.Bag_Status.Reset_Result;
      R #s_Decision_Data.Itm_Data.HBS_Record.PEN_General.Bag_Status.NoDecision;
      R #s_Decision_Data.Itm_Data.HBS_Record.PEN_General.Bag_Status.Pending;
      R #s_Decision_Data.Itm_Data.HBS_Record.PEN_General.Bag_Status.Spare_A;
      R #s_Decision_Data.Itm_Data.HBS_Record.PEN_General.Bag_Status.Spare_B;
      R #s_Decision_Data.Itm_Data.HBS_Record.PEN_General.Bag_Status.Reserved_Signed;
      R #s_Decision_Data.Itm_Data.HBS_Record.PEN_General.Bag_Status.Alarmed;
      R #s_Decision_Data.Itm_Data.HBS_Record.PEN_General.Bag_Status.Cleared;
      R #s_Decision_Data.Itm_Data.HBS_Record.PEN_General.Bag_Status.Communication_Error;
      R #s_Decision_Data.Itm_Data.HBS_Record.PEN_General.Bag_Status.Spare_C;
      R #s_Decision_Data.Itm_Data.HBS_Record.PEN_General.Bag_Status.EDS_Error;
      R #s_Decision_Data.Itm_Data.HBS_Record.PEN_General.Bag_Status.Length_Change;
      R #s_Decision_Data.Itm_Data.HBS_Record.PEN_General.Bag_Status.OOG;
      R #s_Decision_Data.Itm_Data.HBS_Record.PEN_General.Bag_Status.Reinsert;
// Reset other statics/temps
      R #t_Final_Decision_P1;
      R #t_Item_Secure;

      A #s_Decision_Data.Itm_Data.Process_1.EDS_Decision.Cleared_Machine;
      S #s_Decision_Data.Itm_Data.HBS_Record.PEN_General.Bag_Status.Cleared;

      A #s_Decision_Data.Itm_Data.Process_1.EDS_Decision.Cleared_Machine;
      AN #s_Decision_Data.Itm_Data.HBS_Record.PEN_Process_1.Machine_Result_Rcvd;
      JCN NA01;

      L 1;// Update screening status : "CLEAR"
      T #s_Decision_Data.Itm_Data.Process_1.Machine_Result_To_HL;

      SET;
      S #s_Decision_Data.Itm_Data.HBS_Record.PEN_Process_1.Screen_Result.Reached_Screen_Level_1;

NA01:      A #s_Decision_Data.Itm_Data.Process_1.EDS_Decision.Rejected_Machine;
      S #s_Decision_Data.Itm_Data.HBS_Record.PEN_General.Bag_Status.Alarmed;

      A #s_Decision_Data.Itm_Data.Process_1.EDS_Decision.Rejected_Machine;
      AN #s_Decision_Data.Itm_Data.HBS_Record.PEN_Process_1.Machine_Result_Rcvd;
      JCN NA02;

      L 2;// Update screening status : "REJECT"
      T #s_Decision_Data.Itm_Data.Process_1.Machine_Result_To_HL;

      SET;
      S #s_Decision_Data.Itm_Data.HBS_Record.PEN_Process_1.Screen_Result.Failed_Screen_Level_1;

//RTT110 sends only one status from the machine, it can be one of the following:
//Byte1 (Machine Decision)
// - 1 = Machine Threat or Machine Shiled Alarm
// - 2 = Machine Cleared
// - 3 = Machine Analysis Error / Machine Mistrack
// - 4 = Decision Pending
// - 9 = No Scan Bag
NA02:      A #s_Decision_Data.Itm_Data.Process_1.EDS_Decision.Not_Analyzed;//Machine Analysis Error / Machine Mistrack
      JCN NA04;

// PLC log for monitoring purposes
      CALL "FC_Write_Event"
      (  i_Message_ID                := 3892 , // Log: Screening: Not Analyzed
         i_Event_value               := #s_Decision_Data.Itm_Data.LNK ,
         i_DB_Event_Num              := #t_DB_Event_Num_Object ,
         o_Return_Value              := #t_INT_not_used
      );

      L 5;//5=Error unknown
      T #s_Decision_Data.Itm_Data.Process_1.Machine_Result_To_HL;

// Depending on this being a re-screen (depends on current bag status)
      A #t_Bag_ReScreening;
      JCN NA03;
// If 2nd time this bag fails to screen, then reject it
      SET;
      S #s_Decision_Data.Itm_Data.HBS_Record.PEN_General.Bag_Status.Alarmed;
      S #s_Decision_Data.Itm_Data.HBS_Record.PEN_Process_1.Screen_Result.Failed_Screen_Level_1;
      JU NA04;
// Else, just mark as unknown
NA03:      SET;
      S #s_Decision_Data.Itm_Data.HBS_Record.PEN_General.Bag_Status.Unknown;

//EDS_Error
NA04:      A #s_Decision_Data.Itm_Data.Process_1.EDS_Decision.EDS_Error;// EDS_Error (Disposition = 3 on Byte_1)
      AN #s_Decision_Data.Itm_Data.HBS_Record.PEN_Process_1.Machine_Result_Rcvd;
      JCN NA07;

// PLC log for monitoring purposes
      CALL "FC_Write_Event"
      (  i_Message_ID                := 3898 , // Log: Screening: Error
         i_Event_value               := #s_Decision_Data.Itm_Data.LNK ,
         i_DB_Event_Num              := #t_DB_Event_Num_Object ,
         o_Return_Value              := #t_INT_not_used
      );

      L 5;//5=Error unknown
      T #s_Decision_Data.Itm_Data.Process_1.Machine_Result_To_HL;

// Depending on this being a re-screen (depends on current bag status)
      A #t_Bag_ReScreening;
      JCN NA05;
// If 2nd time this bag fails to screen, then reject it
      SET;
      S #s_Decision_Data.Itm_Data.HBS_Record.PEN_General.Bag_Status.Alarmed;
      S #s_Decision_Data.Itm_Data.HBS_Record.PEN_Process_1.Screen_Result.Failed_Screen_Level_1;
      JU NA07;
// Else, just mark as unknown
NA05:      SET;
      S #s_Decision_Data.Itm_Data.HBS_Record.PEN_General.Bag_Status.EDS_Error;

//L2_L3_L4_Unknown
NA07:      A #s_Decision_Data.Itm_Data.Process_1.EDS_Decision.L2_L3_L4_Unknown;// L2_L3_L4_Unknown (Disposition = 3 on Byte_2/3)
      AN #s_Decision_Data.Itm_Data.HBS_Record.PEN_Process_1.Operator_Result_Rcvd;
      AN #t_Decision_Is_L2a;// CPH: For OOG, ignore decision L2a if not Clear
      JCN NA08;
      S #s_Decision_Data.Itm_Data.HBS_Record.PEN_General.Bag_Status.Unknown;

      L 5;// (5=Error unknown)
      T #s_Decision_Data.Itm_Data.Process_1.Operator_Result_To_HL;

NA08:      A #s_Decision_Data.Itm_Data.Process_1.EDS_Decision.L2_Operator_Cleared;// L2 ACCEPT
      AN #s_Decision_Data.Itm_Data.HBS_Record.PEN_Process_1.Operator_Result_Rcvd;
      JCN NA09;// L2 clear
      S #s_Decision_Data.Itm_Data.HBS_Record.PEN_General.Bag_Status.Cleared;

      L 1;// Update screening status : "CLEAR"
      T #s_Decision_Data.Itm_Data.Process_1.Operator_Result_To_HL;

      SET;
      S #s_Decision_Data.Itm_Data.HBS_Record.PEN_Process_1.Screen_Result.Reached_Screen_Level_2;

NA09:      A #s_Decision_Data.Itm_Data.Process_1.EDS_Decision.L2_Operator_Rejected;// L2 REJECT
      AN #s_Decision_Data.Itm_Data.HBS_Record.PEN_Process_1.Operator_Result_Rcvd;
      AN #t_Decision_Is_L2a;// CPH: For OOG, ignore decision L2a if not Clear
      JCN NA10;
      S #s_Decision_Data.Itm_Data.HBS_Record.PEN_General.Bag_Status.Alarmed;

      L 2;// Update screening status : "REJECT"
      T #s_Decision_Data.Itm_Data.Process_1.Operator_Result_To_HL;

      SET;
      S #s_Decision_Data.Itm_Data.HBS_Record.PEN_Process_1.Screen_Result.Failed_Screen_Level_2;

NA10:      A #s_Decision_Data.Itm_Data.Process_1.EDS_Decision.L2_Operator_Timed_Out;
      AN #s_Decision_Data.Itm_Data.HBS_Record.PEN_Process_1.Operator_Result_Rcvd;
      AN #t_Decision_Is_L2a;// CPH: For OOG, ignore decision L2a if not Clear
      JCN NA11;
      S #s_Decision_Data.Itm_Data.HBS_Record.PEN_General.Bag_Status.TimeOut;

      L 4;// Operator Timeout
      T #s_Decision_Data.Itm_Data.Process_1.Operator_Result_To_HL;

//for monitoring purposes
//special reporting number
      CALL "FC_Write_Event"// Log: Screening: L2 Operator Timeout
      (  i_Message_ID                := 3895 , //updated Event list
         i_Event_value               := #s_Decision_Data.Itm_Data.LNK ,
         i_DB_Event_Num              := #t_DB_Event_Num_Object ,
         o_Return_Value              := #t_INT_not_used
      );

NA11:      A #s_Decision_Data.Itm_Data.Process_1.EDS_Decision.L2_Matrix_Timeout_Matrix_Error;
      AN #s_Decision_Data.Itm_Data.HBS_Record.PEN_Process_1.Operator_Result_Rcvd;
      AN #t_Decision_Is_L2a ;// CPH: For OOG, ignore decision L2a if not Clear
      JCN NA12;
      S #s_Decision_Data.Itm_Data.HBS_Record.PEN_General.Bag_Status.Unknown;

      L 5;//Matrix time out (5=Error unknown)
      T #s_Decision_Data.Itm_Data.Process_1.Operator_Result_To_HL;

//special reporting number
      CALL "FC_Write_Event"// Log: Screening: L2 Matrix Timeout
      (  i_Message_ID                := 3893 , //updated Event list
         i_Event_value               := #s_Decision_Data.Itm_Data.LNK ,
         i_DB_Event_Num              := #t_DB_Event_Num_Object ,
         o_Return_Value              := #t_INT_not_used
      );

//IF HIGH THREAT is used, then it should be split into L2/3/4 levels.
//EDS Dispositions: 17, 27, 37 respectively.
//For 06393_LTIA, High Threat is not configured/required. Hence it is not present nor processed in the code.
NA12:      A #s_Decision_Data.Itm_Data.Process_1.EDS_Decision.Obvious_Threat;
      AN #s_Decision_Data.Itm_Data.HBS_Record.PEN_Process_1.Operator_Result_Rcvd;
      JCN NA13;// Obvious threat
      S #s_Decision_Data.Itm_Data.HBS_Record.PEN_General.Bag_Status.Alarmed;

      L 6;
      T #s_Decision_Data.Itm_Data.Process_1.Operator_Result_To_HL;


      SET;
      S #s_Decision_Data.Itm_Data.HBS_Record.PEN_Process_1.Screen_Result.Failed_Screen_Level_2;
//////////////////////////////////////////////////////////////////////////////////////////////////

NA13:      A #s_Decision_Data.Itm_Data.Process_1.EDS_Decision.Decision_Pending;
      JCN NA14;
      S #s_Decision_Data.Itm_Data.HBS_Record.PEN_General.Bag_Status.Pending;

//      L    ???  // Update screening status : "?????"
//      T     #s_Decision_Data.Itm_Data.Process_1.Machine_Result_To_HL
// Requirement is wrong. Machine send s Pending disposition at the exit when still analizing, so another machine decision is sent afterwards.
// So, do not send any report and do not update any result in the BIR.Process1
//      SET
//      S     #s_Decision_Data.Itm_Data.HBS_Record.PEN_Process_1.Screen_Result.Failed_Screen_Level_1// Requirement for CPH: IRS_HBS_RTT110 EDS - 0122


// PLC log for monitoring purposes
      CALL "FC_Write_Event"// Log: Screening: Decision pending
      (  i_Message_ID                := 3897 ,
         i_Event_value               := #s_Decision_Data.Itm_Data.LNK ,
         i_DB_Event_Num              := #t_DB_Event_Num_Object ,
         o_Return_Value              := #t_INT_not_used
      );

// Handle Level 3
NA14:      A #s_Decision_Data.Itm_Data.Process_1.EDS_Decision.L3_Operator_Cleared;// L3 ACCEPT
      AN #s_Decision_Data.Itm_Data.HBS_Record.PEN_Process_1.Operator_Result_Rcvd;
      JCN NA15;
      S #s_Decision_Data.Itm_Data.HBS_Record.PEN_General.Bag_Status.Cleared;

      L 1;// Update screening status : "CLEAR"
      T #s_Decision_Data.Itm_Data.Process_1.Operator_Result_To_HL;

      AN #t_Decision_Is_L2b;
      S #s_Decision_Data.Itm_Data.HBS_Record.PEN_Process_1.Screen_Result.Reached_Screen_Level_3;// L3
      A #t_Decision_Is_L2b;
      S #s_Decision_Data.Itm_Data.HBS_Record.PEN_Process_1.Screen_Result.Reached_Screen_Level_2;// L2b

NA15:      A #s_Decision_Data.Itm_Data.Process_1.EDS_Decision.L3_Operator_Rejected;// L3 REJECT
      AN #s_Decision_Data.Itm_Data.HBS_Record.PEN_Process_1.Operator_Result_Rcvd;
      JCN NA16;
      S #s_Decision_Data.Itm_Data.HBS_Record.PEN_General.Bag_Status.Alarmed;

      L 2;// Update screening status : "REJECT"
      T #s_Decision_Data.Itm_Data.Process_1.Operator_Result_To_HL;

      AN #t_Decision_Is_L2b;
      S #s_Decision_Data.Itm_Data.HBS_Record.PEN_Process_1.Screen_Result.Failed_Screen_Level_3;// L3
      A #t_Decision_Is_L2b;
      S #s_Decision_Data.Itm_Data.HBS_Record.PEN_Process_1.Screen_Result.Failed_Screen_Level_2;// L2b

NA16:      A #s_Decision_Data.Itm_Data.Process_1.EDS_Decision.L3_Operator_Timed_Out;
      AN #s_Decision_Data.Itm_Data.HBS_Record.PEN_Process_1.Operator_Result_Rcvd;
      JCN NA17;
      S #s_Decision_Data.Itm_Data.HBS_Record.PEN_General.Bag_Status.TimeOut;

      L 4;// Operator Timeout
      T #s_Decision_Data.Itm_Data.Process_1.Operator_Result_To_HL;

//for monitoring purposes
//special reporting number
      CALL "FC_Write_Event"// Log: Screening: L3 Operator Timeout
      (  i_Message_ID                := 3896 , //updated Event list
         i_Event_value               := #s_Decision_Data.Itm_Data.LNK ,
         i_DB_Event_Num              := #t_DB_Event_Num_Object ,
         o_Return_Value              := #t_INT_not_used
      );

NA17:      A #s_Decision_Data.Itm_Data.Process_1.EDS_Decision.L3_Matrix_Timeout_Matrix_Error;
      AN #s_Decision_Data.Itm_Data.HBS_Record.PEN_Process_1.Operator_Result_Rcvd;
      JCN NA20;
      S #s_Decision_Data.Itm_Data.HBS_Record.PEN_General.Bag_Status.Unknown;

      L 5;//Matrix time out (5=Error unknown)
      T #s_Decision_Data.Itm_Data.Process_1.Operator_Result_To_HL;

//for monitoring purposes
//special reporting number
      CALL "FC_Write_Event"// Log: Screening: L3 Matrix Timeout
      (  i_Message_ID                := 3894 , //updated Event list
         i_Event_value               := #s_Decision_Data.Itm_Data.LNK ,
         i_DB_Event_Num              := #t_DB_Event_Num_Object ,
         o_Return_Value              := #t_INT_not_used
      );

NA20:      A #s_Decision_Data.Itm_Data.Process_1.EDS_Decision.Not_Analyzed;
      O #s_Decision_Data.Itm_Data.Process_1.EDS_Decision.Decision_Pending;//inasaw ICD-BHS-EDS-0311 ScreeningResult - Disposition Decision pending

      O #s_Decision_Data.Itm_Data.Process_1.EDS_Decision.Cleared_Machine;
      O #s_Decision_Data.Itm_Data.Process_1.EDS_Decision.Rejected_Machine;

      O #s_Decision_Data.Itm_Data.Process_1.EDS_Decision.L2_L3_L4_Unknown;
      O #s_Decision_Data.Itm_Data.Process_1.EDS_Decision.L2_Operator_Cleared;
      O #s_Decision_Data.Itm_Data.Process_1.EDS_Decision.L2_Operator_Rejected;
      O #s_Decision_Data.Itm_Data.Process_1.EDS_Decision.L2_Operator_Timed_Out;
      O #s_Decision_Data.Itm_Data.Process_1.EDS_Decision.L2_Matrix_Timeout_Matrix_Error;

      O #s_Decision_Data.Itm_Data.Process_1.EDS_Decision.L3_Operator_Cleared;
      O #s_Decision_Data.Itm_Data.Process_1.EDS_Decision.L3_Operator_Rejected;
      O #s_Decision_Data.Itm_Data.Process_1.EDS_Decision.L3_Operator_Timed_Out;
      O #s_Decision_Data.Itm_Data.Process_1.EDS_Decision.L3_Matrix_Timeout_Matrix_Error;

      O #s_Decision_Data.Itm_Data.Process_1.EDS_Decision.No_Decision;
      O #s_Decision_Data.Itm_Data.Process_1.EDS_Decision.No_Scan_Bag_RTT;
      O #s_Decision_Data.Itm_Data.Process_1.EDS_Decision.EDS_Error;
      JCN NA99;// In case of new data: Update HBS, LIC and send PackageReport

//ALTIA-1459
//When Message to HL=0 --> below networks will be skipped. It means HBS record will not be updated.
//Result: HBS will have Result_Pending set to TRUE and HBS record will not be updated with latest and legancy information.
      A #s_Decision_Data.Itm_Data.Process_1.EDS_Decision.No_Scan_Bag_RTT;
      JCN NA21;
      R "DB_Pending_Record".THIS[#s_Decision_Data.Itm_Data.PEN_ID].PEN.PEN_Process_1.Result_Pending;

//for monitoring purposes
//special reporting number
      CALL "FC_Write_Event"// Log: Screening: No Scan Item request from BHS
      (  i_Message_ID                := 3899 , //updated Event list
         i_Event_value               := #s_Decision_Data.Itm_Data.LNK ,
         i_DB_Event_Num              := #t_DB_Event_Num_Object ,
         o_Return_Value              := #t_INT_not_used
      );

// Update decision in DB_Pending_Record

NA21:      CALL MOVE
      {value_type := 'Variant'}
      (  IN                          := #s_Decision_Data.Itm_Data.HBS_Record.PEN_Process_1.Screen_Result ,
         OUT                         := "DB_Pending_Record".THIS[#s_Decision_Data.Itm_Data.PEN_ID].PEN.PEN_Process_1.Screen_Result
      );

      CALL MOVE
      {value_type := 'Variant'}
      (  IN                          := #s_Decision_Data.Itm_Data.HBS_Record.PEN_General.Bag_Status ,
         OUT                         := "DB_Pending_Record".THIS[#s_Decision_Data.Itm_Data.PEN_ID].PEN.PEN_General.Bag_Status
      );

// Enable sending of new data if required
      A #s_Decision_Data.Itm_Data.HBS_Record.PEN_Process_1.Update_Send;
      R #s_Decision_Data.Itm_Data.HBS_Record.PEN_Process_1.Update_Send;
      R "DB_Pending_Record".THIS[#s_Decision_Data.Itm_Data.PEN_ID].PEN.PEN_Process_1.Update_Send;

      CALL "FC_Write_Event"   // Screening pending: Update request from HBO
      (  i_Message_ID                := 3814 ,
         i_Event_value               := #s_Decision_Data.Itm_Data.LNK ,
         i_DB_Event_Num              := #t_DB_Event_Num_Object ,
         o_Return_Value              := #t_INT_not_used
      );

// Update decision in DB_HBS_List

      L #s_Decision_Data.Itm_Data.LNK_Record.HBS;
      L 0;
      >I;
      JCN NA22;

      CALL MOVE
      {value_type := 'Variant'}
      (  IN                          := #s_Decision_Data.Itm_Data.HBS_Record.PEN_Process_1 ,
         OUT                         := "DB_HBS_List".HBS[#s_Decision_Data.Itm_Data.LNK_Record.HBS].PEN_Process_1
      );

      CALL MOVE
      {value_type := 'Variant'}
      (  IN                          := #s_Decision_Data.Itm_Data.HBS_Record.PEN_General.Bag_Status ,
         OUT                         := "DB_HBS_List".HBS[#s_Decision_Data.Itm_Data.LNK_Record.HBS].PEN_General.Bag_Status
      );

// Update decision in DB_LIC_List

NA22:      AN #s_Decision_Data.LIC_Missing;
      A(;//condition added from JFKTI-1107. Reason: if LIC is missing, data will be written on LIC[0], which is wrong.
      L #s_Decision_Data.Itm_Data.LNK_Record.LIC;
      L 0;
      >I;
      );
      JCN NA23;

      CALL MOVE
      {value_type := 'Variant'}
      (  IN                          := #s_Decision_Data.Itm_Data.HBS_Record.PEN_Process_1.Screen_Result ,
         OUT                         := "DB_LIC_List".LIC[#s_Decision_Data.Itm_Data.LNK_Record.LIC].BIR.Process_1
      );

      CALL MOVE
      {value_type := 'Variant'}
      (  IN                          := #s_Decision_Data.Itm_Data.HBS_Record.PEN_General.Bag_Status ,
         OUT                         := "DB_LIC_List".LIC[#s_Decision_Data.Itm_Data.LNK_Record.LIC].BIR.Bag_Status
      );


// Determine if more decisions are expected
      CALL "FC_Security_Check"
      (  i_LIC                       := #s_Decision_Data.Itm_Data.LNK_Record.LIC ,
         i_DB_Event_Num              := #t_DB_Event_Num_Object ,
         o_Item_Secure               := #t_Item_Secure
      );

NA23:      A #t_Item_Secure;
      O #s_Decision_Data.Itm_Data.Process_1.EDS_Decision.Not_Analyzed;
      O #s_Decision_Data.Itm_Data.Process_1.EDS_Decision.EDS_Error;
      O #s_Decision_Data.Itm_Data.Process_1.EDS_Decision.L2_L3_L4_Unknown;
      O(;
      A #t_LineType_L1_L2;
      A #t_Decision_Is_L2;
      );
      O(;
      A #t_LineType_L1_L2a_L2b;
      A #t_Decision_Is_L2b;
      );
      O(;
      A #t_LineType_L1_L2_L3;
      A #t_Decision_Is_L3;// L3 is last possible
      );
      S #t_Final_Decision_P1;

      L #s_Decision_Data.Itm_Data.Process_1.Machine_Result_To_HL;
      L 0;
      >I;
      S #s_Decision_Data.Send_Package_Report;
      R #s_Decision_Data.Package_Report_Sent;
      JCN NA24;
      S "DB_Pending_Record".THIS[#s_Decision_Data.Itm_Data.PEN_ID].PEN.PEN_Process_1.Machine_Result_Rcvd;

      A #t_Final_Decision_P1;
      R "DB_Pending_Record".THIS[#s_Decision_Data.Itm_Data.PEN_ID].PEN.PEN_Process_1.Result_Pending;

NA24:      L #s_Decision_Data.Itm_Data.Process_1.Operator_Result_To_HL;
      L 0;
      >I;
      S #s_Decision_Data.Send_Package_Report;
      R #s_Decision_Data.Package_Report_Sent;
      JCN NA25;
      S "DB_Pending_Record".THIS[#s_Decision_Data.Itm_Data.PEN_ID].PEN.PEN_Process_1.Operator_Result_Rcvd;

      A #t_Final_Decision_P1;
      R "DB_Pending_Record".THIS[#s_Decision_Data.Itm_Data.PEN_ID].PEN.PEN_Process_1.Result_Pending;

NA25:      A #s_Decision_Data.Send_Package_Report;
      AN #s_Decision_Data.Package_Report_Sent;
      JCN NA99;

//#nltsal: ALTIA-1369
//Check to determine to which Screening Level does the result belong.
// (Re-arranged for CPH)

      A(;
      L 0;
      L #s_Decision_Data.Itm_Data.Process_1.Machine_Result_To_HL;
      <>I;
      );
      JCN NA26;
      T "DB_HBS_Results".Process_1.Level_1;
      JU NA28;

NA26:      A(;
      L 0;
      L #s_Decision_Data.Itm_Data.Process_1.Operator_Result_To_HL;
      <>I;
      );
      A(;
      A #t_Decision_Is_L2;
      O #t_Decision_Is_L2b;
      O #t_Decision_Is_L2a;
      );
      JCN NA27;
      T "DB_HBS_Results".Process_1.Level_2;
      JU NA28;

NA27:      A(;
      L 0;
      L #s_Decision_Data.Itm_Data.Process_1.Operator_Result_To_HL;
      <>I;
      );
      A #t_Decision_Is_L3;
      JCN NA28;
      T "DB_HBS_Results".Process_1.Level_3;
/////

NA28:      OPN "DB_Send_FIFO";
      L DBNO;
      T #t_INT_not_used;

      CALL MOVE
      {value_type := 'Variant'}
      (  IN                          := #s_Decision_Data.Itm_Data.HBS_Record.PEN_General.Bag_Status ,
         OUT                         := "DB_Pending_Record".THIS[#s_Decision_Data.Itm_Data.PEN_ID].PEN.PEN_General.Bag_Status
      );

      L "DB_Pending_Record".THIS[#t_PEN_ID].PEN.PEN_General.TRA_LNK;
      L 0;
      <>I;
      JCN NA30;

      CALL "FC_Crt_PendingUpd"
      (  i_ID                        := #i_HBO_ID ,
         i_Data                      := #s_Decision_Data.Itm_Data.PEN_ID ,
         i_TRA_LNK                   := "DB_Pending_Record".THIS[#t_PEN_ID].PEN.PEN_General.TRA_LNK ,
         i_FIFO_PLC_DB_num           := #t_INT_not_used ,
         i_DB_Event_Num              := #t_DB_Event_Num_Object ,
         i_Mess_Type                 := 1
      );

NA30:      AN #s_Decision_Data.LIC_Missing;
      JCN NA97;

      L #s_Decision_Data.Itm_Data.LNK_Record.HBS;
      L 0;
      >I;
      JCN NA97;

      CALL MOVE
      {value_type := 'Variant'}
      (  IN                          := "DB_Pending_Record".THIS[#s_Decision_Data.Itm_Data.PEN_ID].PEN.PEN_Process_1 ,
         OUT                         := "DB_HBS_List".HBS[#s_Decision_Data.Itm_Data.LNK_Record.HBS].PEN_Process_1
      );

      CALL "FC_Write_ANY_Record"
      (  i_Record_Number             := #s_Decision_Data.Itm_Data.LNK_Record.LIC ,
         i_ANY_Data_Record           := "DB_UDT_LIC_Record".BIR.Process_1 ,
         i_ANY_Data                  := #s_Decision_Data.Itm_Data.HBS_Record.PEN_Process_1.Screen_Result ,
         i_DB                        := "DB_LIC_List" ,
         i_DB_Event_Num              := #t_DB_Event_Num_Object
      );

      CALL "FC_Write_Event"
      (  i_Message_ID                := 1210 , // Send PackageReport: Screening Result
         i_Event_value               := #s_Decision_Data.Itm_Data.LNK ,
         i_DB_Event_Num              := #t_DB_Event_Num_Object ,
         o_Return_Value              := #t_INT_not_used
      );

      JU NA98;

NA97:      CALL "FC_Crt_PackScrnPen"
      (  i_ID                        := #i_HBO_ID ,
         i_PEN_ID                    := #s_Decision_Data.Itm_Data.PEN_ID ,
         i_FIFO_PLC_DB_num           := #t_INT_not_used ,
         i_DB_Event_Num              := #t_DB_Event_Num_Object
      );

NA98:      SET;
      S #s_Decision_Data.Package_Report_Sent;

NA99:      NOP 0;
NETWORK
TITLE = OA: Update PROCESS_1 statisticals upon decision or timeout

      A #s_OS_New_Decision_Avail;
      AN #i_Test_Mode_Active;// Don't update machine decision statisticals in test mode
      JCN OA99;

      A #s_Decision_Data.Itm_Data.Process_1.EDS_Decision.Cleared_Machine;
      JCN OA02;

      L #s_Statisticals.R1.Count_Cleared;
      L 1;
      +I;
      JP OA01;
      L 1;
OA01:      T #s_Statisticals.R1.Count_Cleared;

      JU OA99;
OA02:      A #s_Decision_Data.Itm_Data.Process_1.EDS_Decision.Rejected_Machine;
      JCN OA04;

      L #s_Statisticals.R1.Count_Rejected;
      L 1;
      +I;
      JP OA03;
      L 1;
OA03:      T #s_Statisticals.R1.Count_Rejected;
      JU OA99;

OA04:      A #s_Decision_Data.Itm_Data.Process_1.EDS_Decision.Not_Analyzed;
      JCN OA06;

      L #s_Statisticals.R1.Count_NotAnalyzed;
      L 1;
      +I;
      JP OA05;
      L 1;
OA05:      T #s_Statisticals.R1.Count_NotAnalyzed;

      JU OA99;
OA06:      A #s_Decision_Data.Itm_Data.Process_1.EDS_Decision.L2_Operator_Cleared;// Evaluate L2 (operator) decision
      JCN OA08;// L2 clear

      L #s_Statisticals.R2.Count_Cleared;
      L 1;
      +I;
      JP OA07;
      L 1;
OA07:      T #s_Statisticals.R2.Count_Cleared;
      JU OA99;

OA08:      A #s_Decision_Data.Itm_Data.Process_1.EDS_Decision.L2_Operator_Rejected;// L2 fail
      JCN OA10;

      L #s_Statisticals.R2.Count_Rejected;
      L 1;
      +I;
      JP OA09;
      L 1;
OA09:      T #s_Statisticals.R2.Count_Rejected;

      JU OA99;

OA10:      A #s_Decision_Data.Itm_Data.Process_1.EDS_Decision.L2_Operator_Timed_Out;
      JCN OA12;

      L #s_Statisticals.R2.Count_TimeOut;
      L 1;
      +I;
      JP OA11;
      L 1;
OA11:      T #s_Statisticals.R2.Count_TimeOut;

      JU OA99;

OA12:      A #s_Decision_Data.Itm_Data.Process_1.EDS_Decision.L2_Matrix_Timeout_Matrix_Error;
      JCN OA14;

      L #s_Statisticals.R2.Matrix_Timeout;
      L 1;
      +I;
      JP OA13;
      L 1;
OA13:      T #s_Statisticals.R2.Matrix_Timeout;

      JU OA99;

OA14:      A #s_Decision_Data.Itm_Data.Process_1.EDS_Decision.L3_Operator_Cleared;// Evaluate L3 (operator) decision
      JCN OA16;// L2 clear

      L #s_Statisticals.R3.Count_Cleared;
      L 1;
      +I;
      JP OA15;
      L 1;
OA15:      T #s_Statisticals.R3.Count_Cleared;
      JU OA99;

OA16:      A #s_Decision_Data.Itm_Data.Process_1.EDS_Decision.L3_Operator_Rejected;// L3 fail
      JCN OA18;

      L #s_Statisticals.R3.Count_Rejected;
      L 1;
      +I;
      JP OA17;
      L 1;
OA17:      T #s_Statisticals.R3.Count_Rejected;

      JU OA99;

OA18:      A #s_Decision_Data.Itm_Data.Process_1.EDS_Decision.L3_Operator_Timed_Out;
      JCN OA20;

      L #s_Statisticals.R3.Count_TimeOut;
      L 1;
      +I;
      JP OA19;
      L 1;
OA19:      T #s_Statisticals.R3.Count_TimeOut;

      JU OA99;

OA20:      A #s_Decision_Data.Itm_Data.Process_1.EDS_Decision.L3_Matrix_Timeout_Matrix_Error;
      JCN OA99;

      L #s_Statisticals.R3.Matrix_Timeout;
      L 1;
      +I;
      JP OA21;
      L 1;
OA21:      T #s_Statisticals.R3.Matrix_Timeout;

OA99:      NOP 0;
NETWORK
TITLE = PA: Force reject (Not supported)
//When a bag decision is pending while it's no longer required. The bag will be
//force rejected
      CALL #s_FB_HBS_Force_Reject
      (  i_ID                        := #i_HBO_ID ,
         i_Forced_Reject_Ack         := #i_IO_Forced_Reject_Ack ,
         o_Force_Reject              := #o_IO_Force_Reject ,
         o_Pseudo_Code_ForceRej      := #o_IO_Pseud_Code_ForceRej
      );

      A #o_IO_Force_Reject;
      FP #s_FP_Force_Reject;
      JCN PA99;

      L #s_Statisticals.Force_Rejected;
      L 1;
      +I;
      JP PA01;
      L 1;
PA01:      T #s_Statisticals.Force_Rejected;

PA99:      NOP 0;
NETWORK
TITLE = QA: Send and clear statisticals
      A #i_CMD_Send_Stat;
      JCN QA99;

      CALL "FC_Write_Event"
      (  i_Message_ID                := 2001 ,
         i_Event_value               := #s_Statisticals.Bags_Handed_Over ,
         i_DB_Event_Num              := #t_DB_Event_Num_Object ,
         o_Return_Value              := #t_INT_not_used
      );

      CALL "FC_Write_Event"
      (  i_Message_ID                := 2002 ,
         i_Event_value               := #s_Statisticals.Tracking.Positively_Tracked ,
         i_DB_Event_Num              := #t_DB_Event_Num_Object ,
         o_Return_Value              := #t_INT_not_used
      );

      CALL "FC_Write_Event"
      (  i_Message_ID                := 2003 ,
         i_Event_value               := #s_Statisticals.Tracking.Trk_Lost_Result_Pending ,
         i_DB_Event_Num              := #t_DB_Event_Num_Object ,
         o_Return_Value              := #t_INT_not_used
      );

      CALL "FC_Write_Event"
      (  i_Message_ID                := 2004 ,
         i_Event_value               := #s_Statisticals.Tracking.Trk_Lost_No_Result ,
         i_DB_Event_Num              := #t_DB_Event_Num_Object ,
         o_Return_Value              := #t_INT_not_used
      );

      CALL "FC_Write_Event"
      (  i_Message_ID                := 2005 ,
         i_Event_value               := #s_Statisticals.R1.No_Decision_Required ,
         i_DB_Event_Num              := #t_DB_Event_Num_Object ,
         o_Return_Value              := #t_INT_not_used
      );

      CALL "FC_Write_Event"
      (  i_Message_ID                := 2006 ,
         i_Event_value               := #s_Statisticals.R1.Count_Cleared ,
         i_DB_Event_Num              := #t_DB_Event_Num_Object ,
         o_Return_Value              := #t_INT_not_used
      );

      CALL "FC_Write_Event"
      (  i_Message_ID                := 2007 ,
         i_Event_value               := #s_Statisticals.R1.Count_Rejected ,
         i_DB_Event_Num              := #t_DB_Event_Num_Object ,
         o_Return_Value              := #t_INT_not_used
      );

      CALL "FC_Write_Event"
      (  i_Message_ID                := 2008 ,
         i_Event_value               := #s_Statisticals.R2.Count_Cleared ,
         i_DB_Event_Num              := #t_DB_Event_Num_Object ,
         o_Return_Value              := #t_INT_not_used
      );

      CALL "FC_Write_Event"
      (  i_Message_ID                := 2009 ,
         i_Event_value               := #s_Statisticals.R2.Count_Rejected ,
         i_DB_Event_Num              := #t_DB_Event_Num_Object ,
         o_Return_Value              := #t_INT_not_used
      );

      CALL "FC_Write_Event"
      (  i_Message_ID                := 2010 ,
         i_Event_value               := #s_Statisticals.R2.Count_TimeOut ,
         i_DB_Event_Num              := #t_DB_Event_Num_Object ,
         o_Return_Value              := #t_INT_not_used
      );

      CALL "FC_Write_Event"
      (  i_Message_ID                := 2011 ,
         i_Event_value               := #s_Statisticals.R1.Count_NotAnalyzed ,
         i_DB_Event_Num              := #t_DB_Event_Num_Object ,
         o_Return_Value              := #t_INT_not_used
      );

      CALL "FC_Write_Event"
      (  i_Message_ID                := 2012 ,
         i_Event_value               := #s_Statisticals.Force_Rejected ,
         i_DB_Event_Num              := #t_DB_Event_Num_Object ,
         o_Return_Value              := #t_INT_not_used
      );


      CALL "FC_Write_Event"
      (  i_Message_ID                := 2013 ,
         i_Event_value               := #s_Statisticals.R2.Matrix_Timeout ,
         i_DB_Event_Num              := #t_DB_Event_Num_Object ,
         o_Return_Value              := #t_INT_not_used
      );

//Added extra for RTT110
      CALL "FC_Write_Event"
      (  i_Message_ID                := 2014 ,
         i_Event_value               := #s_Statisticals.R3.Count_Cleared ,
         i_DB_Event_Num              := #t_DB_Event_Num_Object ,
         o_Return_Value              := #t_INT_not_used
      );

      CALL "FC_Write_Event"
      (  i_Message_ID                := 2015 ,
         i_Event_value               := #s_Statisticals.R3.Count_Rejected ,
         i_DB_Event_Num              := #t_DB_Event_Num_Object ,
         o_Return_Value              := #t_INT_not_used
      );

      CALL "FC_Write_Event"
      (  i_Message_ID                := 2016 ,
         i_Event_value               := #s_Statisticals.R3.Count_TimeOut ,
         i_DB_Event_Num              := #t_DB_Event_Num_Object ,
         o_Return_Value              := #t_INT_not_used
      );

      CALL "FC_Write_Event"
      (  i_Message_ID                := 2017 ,
         i_Event_value               := #s_Statisticals.R3.Matrix_Timeout ,
         i_DB_Event_Num              := #t_DB_Event_Num_Object ,
         o_Return_Value              := #t_INT_not_used
      );
////////////////////

// IF Sample type such that counters need to be reset,
      A(;
      L "DB_Setting".common.Sample_Type_Stat_Counters;
      L 2;// CUMULATIVE
      ==I;
      );
      JCN QA99;
// THEN reset values.
      L 0;
      T #s_Statisticals.Bags_Handed_Over;
      T #s_Statisticals.R1.Count_Cleared;
      T #s_Statisticals.R2.Count_Cleared;
      T #s_Statisticals.R3.Count_Cleared;
      T #s_Statisticals.R1.Count_Rejected;
      T #s_Statisticals.R2.Count_Rejected;
      T #s_Statisticals.R3.Count_Rejected;
      T #s_Statisticals.R1.Count_NotAnalyzed;
      T #s_Statisticals.R2.Count_TimeOut;
      T #s_Statisticals.R3.Count_TimeOut;
      T #s_Statisticals.R2.Matrix_Timeout;
      T #s_Statisticals.R3.Matrix_Timeout;
      T #s_Statisticals.Tracking.Positively_Tracked;
      T #s_Statisticals.Tracking.Trk_Lost_Result_Pending;
      T #s_Statisticals.Tracking.Trk_Lost_No_Result;
      T #s_Statisticals.Force_Rejected;
      T #s_Statisticals.R1.No_Decision_Required;

QA99:      NOP 0;
NETWORK
TITLE = RA: Date/Time Master Clock Designator
      CLR;// RTT is master clock
      = #o_IO_MasterClkDesignator;// No need to send BHS clock

      L #i_IO_Time_Sync_Sec;// Seconds [00..59]
      T #o_IO_Time_Sync_Sec;

      L #i_IO_Time_Sync_Min;// Minutes [00..59]
      T #o_IO_Time_Sync_Min;

      L #i_IO_Time_Sync_Hour;// Time_hours [01..24]
      T #o_IO_Time_Sync_Hour;

      L #i_IO_Time_Sync_Day;// Day of month [1..31]
      T #o_IO_Time_Sync_Day;

      L #i_IO_Time_Sync_Month;// Month [1..31]
      T #o_IO_Time_Sync_Month;

      L #i_IO_Time_Sync_Year;// Year  [0..99]
      T #o_IO_Time_Sync_Year;

NETWORK
TITLE = SA: Object/Section states
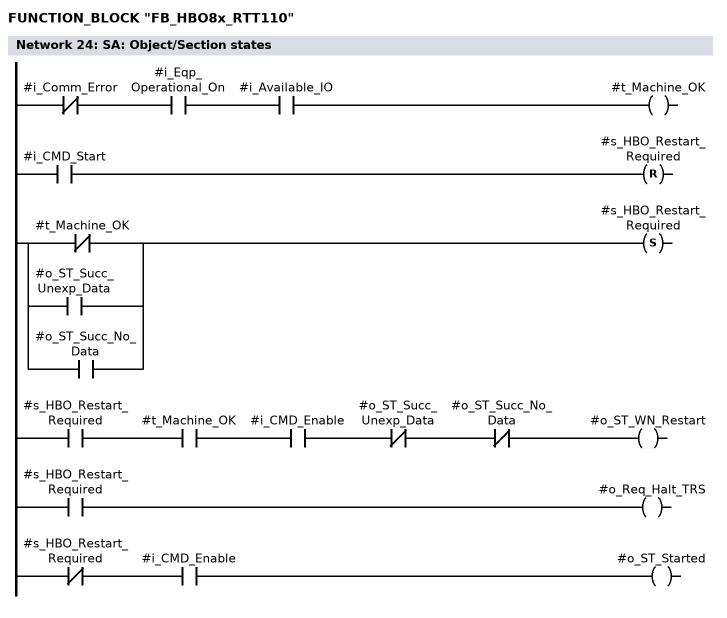
      AN #i_Comm_Error;
      A #i_Eqp_Operational_On;
      A #i_Available_IO;
      = #t_Machine_OK;

      A #i_CMD_Start;
      R #s_HBO_Restart_Required;

      AN #t_Machine_OK;
      O #o_ST_Succ_Unexp_Data;
      O #o_ST_Succ_No_Data;
      S #s_HBO_Restart_Required;

      A #s_HBO_Restart_Required;
      A #t_Machine_OK;
      A #i_CMD_Enable;
      AN #o_ST_Succ_Unexp_Data;
      AN #o_ST_Succ_No_Data;
      = #o_ST_WN_Restart;

      A #s_HBO_Restart_Required;
      = #o_Req_Halt_TRS;

      AN #s_HBO_Restart_Required;
      A #i_CMD_Enable;
      = #o_ST_Started;
NETWORK
TITLE = TA: Copy BHS_ID.BAGIDARRAY (Data + IATA + PSEUDO) to output
//BHS_ID = BagIDArray + IATA + PSEUDO
      TAR2 #t_AR2_Store_Restore;// AR2 Store

      L P##i_IO_BHS_ID;// 'area-crossing pointer'
      L #t_Base_Address;// 'relative address'-mask
      +D;
      LAR1;// 'absolute address' Source
      LAR2 P##t_IO_BHS_ID;//  address Destination

      L W[ AR1, P#0.0];// Copy ANY pointer
      T LW[ AR2, P#0.0];// Byte0=$10 (for S7), Byte1=data type
      L W[ AR1, P#2.0];
      T LW[ AR2, P#2.0];// Byte2..3=Repetition factor
      L W[ AR1, P#4.0];
      T LW[ AR2, P#4.0];// Byte4..5=DB number
      L D[ AR1, P#6.0];
      T LD[ AR2, P#6.0];// Byte6=memory area, Byte7..9=Byte,Bit address

      LAR2 #t_AR2_Store_Restore;// AR2 Restore

      CALL BLKMOV
      {blk_type := 'Variant'}
      (  SRCBLK                      := #s_BHS_ID ,
         RET_VAL                     := #t_INT_not_used ,
         DSTBLK                      := #t_IO_BHS_ID
      );

NETWORK
TITLE = UA: Log (1:) BHS.Infeed Bag Process to ApplicationLog
//Log the screening raw data message to the ApplicationLog

      A #o_IO_Inf_Bag_Data_Ready;
      FP #s_FP_IO_Inf_Bag_Data_Ready;
      JCN UA99;

// Clear temp LogMessage using "DB_Outgoing_Msgs".Logging.MessageBody which cleared after usage
      CALL BLKMOV
      {blk_type := 'Variant'}
      (  SRCBLK                      := "DB_Outgoing_Msgs".Logging.MessageBody ,
         RET_VAL                     := #t_INT_not_used ,
         DSTBLK                      := #t_LogMessage
      );


// Add Prefix and separator to log message for indication which message is logged
// '1:' = BHS.Infeed Bag Process
      L '1';
      T #t_LogMessage.Prefix;
      L ':';
      T #t_LogMessage.Separator;

// Convert raw data to a string of ASCII characters
      CALL "FC_Any_Hex_To_Any_ASCII"
      (  i_ANY_Hex_Src               := #s_BHS_ID ,
         i_ANY_ASCII_Dst             := #t_LogMessage.MessageBody ,
         i_DB_Event_Num              := #t_DB_Event_Num_Object
      );


// Load the complete message into Outgoing message buffer
      CALL BLKMOV
      {blk_type := 'Variant'}
      (  SRCBLK                      := #t_LogMessage ,
         RET_VAL                     := #t_INT_not_used ,
         DSTBLK                      := "DB_Outgoing_Msgs".Logging.MessageBody
      );



// Send 2602 ApplicationLog Message
      CALL "FC_Snd_Log_Txt_Msg"
      (  i_ID                        := #i_HBO_ID ,
         i_Event_value               := 1
      );

UA99:      NOP 0;

NETWORK
TITLE = UB:Log(2:) EDS.Exit Bag Process to ApplicationLog

//Log the screening raw data message to the ApplicationLog

      A #i_IO_Receive_Data_Outf;
      FP #s_FP_IO_Receive_Data_Outf;
      JCN UB99;

// Clear temp LogMessage using "DB_Outgoing_Msgs".Logging.MessageBody which cleared after usage
      CALL BLKMOV
      {blk_type := 'Variant'}
      (  SRCBLK                      := "DB_Outgoing_Msgs".Logging.MessageBody ,
         RET_VAL                     := #t_INT_not_used ,
         DSTBLK                      := #t_LogMessage
      );

// Add Prefix and separator to log message for indication which message is logged
// '2:' = EDS.Exit Bag Process
      L '2';
      T #t_LogMessage.Prefix;
      L ':';
      T #t_LogMessage.Separator;

// Convert raw data to a string of ASCII characters
      CALL "FC_Any_Hex_To_Any_ASCII"
      (  i_ANY_Hex_Src               := #s_ISD_ID_Tracking ,
         i_ANY_ASCII_Dst             := #t_LogMessage.MessageBody ,
         i_DB_Event_Num              := #t_DB_Event_Num_Object
      );

// Load the complete message into Outgoing message buffer
      CALL BLKMOV
      {blk_type := 'Variant'}
      (  SRCBLK                      := #t_LogMessage ,
         RET_VAL                     := #t_INT_not_used ,
         DSTBLK                      := "DB_Outgoing_Msgs".Logging.MessageBody
      );


// Send 2602 ApplicationLog Message
      CALL "FC_Snd_Log_Txt_Msg"
      (  i_ID                        := #i_HBO_ID ,
         i_Event_value               := 2
      );


UB99:      NOP 0;

NETWORK
TITLE = UC:Log(3:) EDS.Screening Result to ApplicationLog
//Log the screening raw data message to the ApplicationLog
      A #i_IO_Decision_Available;
      FP #s_FP_IO_Decision_Available;
      JCN UC99;

// Clear temp LogMessage using "DB_Outgoing_Msgs".Logging.MessageBody which cleared after usage
      CALL BLKMOV
      {blk_type := 'Variant'}
      (  SRCBLK                      := "DB_Outgoing_Msgs".Logging.MessageBody ,
         RET_VAL                     := #t_INT_not_used ,
         DSTBLK                      := #t_LogMessage
      );

// Add Prefix and separator to log message for indication which message is logged
// '3:' = EDS.Screening Result
      L '3';
      T #t_LogMessage.Prefix;
      L ':';
      T #t_LogMessage.Separator;

// Convert raw data to a string of ASCII characters
      CALL "FC_Any_Hex_To_Any_ASCII"
      (  i_ANY_Hex_Src               := #s_ISD_ID_Decision ,
         i_ANY_ASCII_Dst             := #t_LogMessage.MessageBody ,
         i_DB_Event_Num              := #t_DB_Event_Num_Object
      );


// Load the complete message into Outgoing message buffer
      CALL BLKMOV
      {blk_type := 'Variant'}
      (  SRCBLK                      := #t_LogMessage ,
         RET_VAL                     := #t_INT_not_used ,
         DSTBLK                      := "DB_Outgoing_Msgs".Logging.MessageBody
      );


// Send 2602 ApplicationLog Message
      CALL "FC_Snd_Log_Txt_Msg"
      (  i_ID                        := #i_HBO_ID ,
         i_Event_value               := 3
      );

UC99:      NOP 0;

NETWORK
TITLE = UD:Log(4:) BHS.ForcedReject to ApplicationLog

//Log the screening raw data message to the ApplicationLog

      A #o_IO_Force_Reject;
      FP #s_FP_IO_Force_Reject;
      JCN UD99;

// Clear temp LogMessage using "DB_Outgoing_Msgs".Logging.MessageBody which cleared after usage
      CALL BLKMOV
      {blk_type := 'Variant'}
      (  SRCBLK                      := "DB_Outgoing_Msgs".Logging.MessageBody ,
         RET_VAL                     := #t_INT_not_used ,
         DSTBLK                      := #t_LogMessage
      );

// Add Prefix and separator to log message for indication which message is logged
// '4:' = BHS.ForcedReject
      L '4';
      T #t_LogMessage.Prefix;
      L ':';
      T #t_LogMessage.Separator;

// Convert raw data to a string of ASCII characters
      CALL "FC_Any_Hex_To_Any_ASCII"
      (  i_ANY_Hex_Src               := #o_IO_Pseud_Code_ForceRej ,
         i_ANY_ASCII_Dst             := #t_LogMessage.MessageBody ,
         i_DB_Event_Num              := #t_DB_Event_Num_Object
      );

// Load the complete message into Outgoing message buffer
      CALL BLKMOV
      {blk_type := 'Variant'}
      (  SRCBLK                      := #t_LogMessage ,
         RET_VAL                     := #t_INT_not_used ,
         DSTBLK                      := "DB_Outgoing_Msgs".Logging.MessageBody
      );


// Send 2602 ApplicationLog Message
      CALL "FC_Snd_Log_Txt_Msg"
      (  i_ID                        := #i_HBO_ID ,
         i_Event_value               := 4
      );


UD99:      NOP 0;


NETWORK
TITLE = UE:Log(5:) EDS.ForcedReject to ApplicationLog

//Log the screening raw data message to the ApplicationLog

      A #i_IO_Forced_Reject_Ack;
      FP #s_FP_IO_Forced_Reject_Ack;
      JCN UE99;

// Clear temp LogMessage using "DB_Outgoing_Msgs".Logging.MessageBody which cleared after usage
      CALL BLKMOV
      {blk_type := 'Variant'}
      (  SRCBLK                      := "DB_Outgoing_Msgs".Logging.MessageBody ,
         RET_VAL                     := #t_INT_not_used ,
         DSTBLK                      := #t_LogMessage
      );


// Add Prefix and separator to log message for indication which message is logged
// '5:' = EDS.ForcedReject
      L '5';
      T #t_LogMessage.Prefix;
      L ':';
      T #t_LogMessage.Separator;

// Convert raw data to a string of ASCII characters
      CALL "FC_Any_Hex_To_Any_ASCII"
      (  i_ANY_Hex_Src               := #s_ISD_ID_Decision ,
         i_ANY_ASCII_Dst             := #t_LogMessage.MessageBody ,
         i_DB_Event_Num              := #t_DB_Event_Num_Object
      );

// Load the complete message into Outgoing message buffer
      CALL BLKMOV
      {blk_type := 'Variant'}
      (  SRCBLK                      := #t_LogMessage ,
         RET_VAL                     := #t_INT_not_used ,
         DSTBLK                      := "DB_Outgoing_Msgs".Logging.MessageBody
      );

// Send 2602 ApplicationLog Message
      CALL "FC_Snd_Log_Txt_Msg"
      (  i_ID                        := #i_HBO_ID ,
         i_Event_value               := 5
      );


UE99:      NOP 0;

END_FUNCTION_BLOCK
